C03639=1044.322,83.041,413.959,170.198,36.682,156.905
C03640=1044.329,83.290,413.941,170.200,36.684,156.905
C03641=1044.335,83.539,413.922,170.201,36.685,156.905
C03642=1044.341,83.788,413.904,170.203,36.687,156.906
C03643=1044.347,84.037,413.885,170.205,36.688,156.906
C03644=1044.353,84.287,413.866,170.206,36.689,156.906
C03645=1044.359,84.536,413.848,170.208,36.690,156.906
C03646=1044.366,84.785,413.829,170.211,36.692,156.906
C03647=1044.372,85.034,413.811,170.212,36.693,156.907
C03648=1044.378,85.284,413.791,170.214,36.694,156.907
C03649=1044.384,85.533,413.773,170.216,36.695,156.907
C03650=1044.391,85.782,413.754,170.217,36.697,156.907
C03651=1044.397,86.031,413.735,170.219,36.699,156.908
C03652=1044.403,86.280,413.716,170.222,36.700,156.908
C03653=1044.409,86.529,413.697,170.223,36.701,156.908
C03654=1044.416,86.779,413.679,170.225,36.702,156.909
C03655=1044.422,87.028,413.660,170.227,36.704,156.909
C03656=1044.428,87.277,413.641,170.229,36.705,156.909
C03657=1044.434,87.526,413.622,170.230,36.706,156.909
C03658=1044.440,87.775,413.604,170.233,36.707,156.909
C03659=1044.447,88.024,413.585,170.235,36.709,156.910
C03660=1044.453,88.274,413.566,170.236,36.710,156.910
C03661=1044.459,88.523,413.547,170.238,36.711,156.910
C03662=1044.466,88.773,413.528,170.240,36.712,156.910
C03663=1044.472,89.022,413.509,170.241,36.713,156.911
C03664=1044.479,89.271,413.491,170.243,36.715,156.911
C03665=1044.485,89.521,413.471,170.246,36.717,156.911
C03666=1044.491,89.770,413.453,170.248,36.718,156.912
C03667=1044.497,90.019,413.434,170.249,36.719,156.912
C03668=1044.504,90.268,413.416,170.251,36.720,156.912
C03669=1044.510,90.517,413.396,170.253,36.722,156.912
C03670=1044.516,90.766,413.376,170.254,36.723,156.913
C03671=1044.522,91.015,413.358,170.257,36.724,156.913
C03672=1044.528,91.265,413.338,170.259,36.726,156.913
C03673=1044.534,91.514,413.320,170.260,36.727,156.913
C03674=1044.540,91.763,413.301,170.262,36.728,156.914
C03675=1044.547,92.012,413.281,170.264,36.730,156.914
C03676=1044.552,92.261,413.262,170.265,36.731,156.914
C03677=1044.559,92.510,413.243,170.268,36.733,156.914
C03678=1044.564,92.760,413.224,170.270,36.734,156.915
C03679=1044.572,93.045,413.202,170.272,36.735,156.915
C03680=1044.579,93.332,413.180,170.274,36.737,156.915
C03681=1044.586,93.617,413.158,170.276,36.738,156.916
C03682=1044.593,93.904,413.136,170.278,36.740,156.916
C03683=1044.599,94.153,413.117,170.280,36.741,156.916
C03684=1044.606,94.402,413.098,170.282,36.743,156.916
C03685=1044.612,94.651,413.078,170.284,36.744,156.917
C03686=1044.618,94.900,413.060,170.285,36.745,156.917
C03687=1044.624,95.150,413.040,170.287,36.747,156.917
C03688=1044.630,95.398,413.021,170.290,36.748,156.917
C03689=1044.636,95.648,413.002,170.291,36.749,156.918
C03690=1044.643,95.897,412.983,170.293,36.751,156.918
C03691=1044.649,96.146,412.963,170.295,36.752,156.918
C03692=1044.655,96.396,412.944,170.296,36.753,156.918
C03693=1044.661,96.645,412.925,170.298,36.755,156.919
C03694=1044.667,96.894,412.905,170.301,36.756,156.919
C03695=1044.674,97.143,412.886,170.302,36.758,156.919
C03696=1044.679,97.392,412.867,170.304,36.759,156.920
C03697=1044.686,97.641,412.848,170.306,36.760,156.920
C03698=1044.692,97.891,412.828,170.308,36.761,156.920
C03699=1044.699,98.140,412.809,170.309,36.763,156.920
C03700=1044.705,98.389,412.789,170.312,36.764,156.921
C03701=1044.710,98.638,412.770,170.314,36.766,156.921
C03702=1044.717,98.887,412.751,170.315,36.767,156.921
C03703=1044.723,99.136,412.732,170.317,36.768,156.921
C03704=1044.730,99.386,412.713,170.319,36.769,156.922
C03705=1044.736,99.635,412.693,170.321,36.771,156.922
C03706=1044.742,99.884,412.674,170.322,36.772,156.922
C03707=1044.748,100.133,412.654,170.325,36.774,156.922
C03708=1044.755,100.382,412.635,170.327,36.775,156.923
C03709=1044.761,100.631,412.615,170.328,36.776,156.923
C03710=1044.767,100.881,412.596,170.330,36.777,156.923
C03711=1044.773,101.130,412.576,170.332,36.779,156.923
C03712=1044.779,101.379,412.557,170.334,36.780,156.924
C03713=1044.785,101.628,412.537,170.336,36.782,156.924
C03714=1044.791,101.877,412.518,170.338,36.783,156.924
C03715=1044.798,102.127,412.498,170.340,36.785,156.925
C03716=1044.803,102.376,412.478,170.341,36.786,156.925
C03717=1044.809,102.625,412.458,170.343,36.787,156.925
C03718=1044.816,102.874,412.440,170.346,36.788,156.925
C03719=1044.822,103.123,412.420,170.347,36.790,156.926
C03720=1044.828,103.372,412.400,170.349,36.792,156.926
C03721=1044.834,103.622,412.380,170.351,36.793,156.926
C03722=1044.840,103.870,412.360,170.352,36.794,156.926
C03723=1044.846,104.120,412.341,170.354,36.796,156.927
C03724=1044.853,104.368,412.322,170.357,36.797,156.927
C03725=1044.859,104.618,412.301,170.359,36.798,156.927
C03726=1044.865,104.867,412.282,170.360,36.800,156.928
C03727=1044.871,105.116,412.262,170.362,36.801,156.928
C03728=1044.877,105.365,412.242,170.364,36.803,156.928
C03729=1044.883,105.615,412.223,170.365,36.804,156.928
C03730=1044.890,105.864,412.203,170.368,36.805,156.929
C03731=1044.896,106.112,412.183,170.370,36.807,156.929
C03732=1044.901,106.362,412.164,170.371,36.808,156.929
C03733=1044.908,106.611,412.144,170.373,36.810,156.929
C03734=1044.914,106.860,412.124,170.375,36.811,156.930
C03735=1044.920,107.110,412.105,170.377,36.812,156.930
C03736=1044.927,107.358,412.085,170.379,36.814,156.930
C03737=1044.933,107.608,412.065,170.381,36.815,156.931
C03738=1044.939,107.857,412.046,170.383,36.816,156.931
C03739=1044.945,108.106,412.026,170.385,36.818,156.931
C03740=1044.951,108.355,412.005,170.386,36.819,156.931
C03741=1044.957,108.604,411.985,170.389,36.821,156.932
C03742=1044.963,108.854,411.966,170.391,36.822,156.932
C03743=1044.971,109.139,411.944,170.393,36.824,156.932
C03744=1044.977,109.425,411.921,170.395,36.825,156.933
C03745=1044.986,109.711,411.897,170.397,36.827,156.933
C03746=1044.992,109.997,411.874,170.400,36.828,156.933
C03747=1044.998,110.247,411.855,170.401,36.829,156.933
C03748=1045.005,110.495,411.836,170.403,36.831,156.934
C03749=1045.011,110.745,411.816,170.405,36.832,156.934
C03750=1045.017,110.993,411.796,170.407,36.834,156.934
C03751=1045.023,111.242,411.776,170.408,36.835,156.934
C03752=1045.030,111.492,411.755,170.411,36.837,156.935
C03753=1045.036,111.741,411.736,170.413,36.838,156.935
C03754=1045.042,111.990,411.716,170.414,36.839,156.935
C03755=1045.048,112.240,411.696,170.416,36.840,156.936
C03756=1045.054,112.488,411.676,170.418,36.842,156.936
C03757=1045.060,112.737,411.656,170.420,36.843,156.936
C03758=1045.067,112.987,411.636,170.422,36.845,156.936
C03759=1045.073,113.235,411.616,170.424,36.847,156.937
C03760=1045.078,113.485,411.595,170.426,36.848,156.937
C03761=1045.085,113.734,411.575,170.428,36.849,156.937
C03762=1045.091,113.983,411.555,170.429,36.851,156.938
C03763=1045.097,114.232,411.535,170.432,36.852,156.938
C03764=1045.103,114.481,411.514,170.434,36.853,156.938
C03765=1045.108,114.730,411.494,170.435,36.855,156.939
C03766=1045.114,114.979,411.474,170.437,36.856,156.939
C03767=1045.121,115.229,411.454,170.439,36.858,156.939
C03768=1045.127,115.478,411.434,170.442,36.859,156.939
C03769=1045.132,115.727,411.413,170.443,36.861,156.940
C03770=1045.139,115.976,411.393,170.445,36.863,156.940
C03771=1045.145,116.225,411.373,170.447,36.864,156.940
C03772=1045.150,116.474,411.352,170.448,36.866,156.941
C03773=1045.157,116.724,411.332,170.450,36.867,156.941
C03774=1045.163,116.972,411.312,170.453,36.868,156.941
C03775=1045.169,117.222,411.292,170.455,36.870,156.941
C03776=1045.175,117.471,411.271,170.456,36.871,156.942
C03777=1045.181,117.719,411.250,170.458,36.873,156.942
C03778=1045.187,117.969,411.230,170.460,36.874,156.942
C03779=1045.193,118.218,411.210,170.463,36.875,156.943
C03780=1045.199,118.467,411.190,170.464,36.877,156.943
C03781=1045.205,118.716,411.169,170.466,36.879,156.943
C03782=1045.211,118.965,411.149,170.468,36.880,156.943
C03783=1045.217,119.215,411.128,170.470,36.882,156.944
C03784=1045.223,119.463,411.108,170.472,36.883,156.944
C03785=1045.229,119.712,411.088,170.474,36.885,156.944
C03786=1045.235,119.962,411.067,170.476,36.886,156.945
C03787=1045.241,120.210,411.047,170.477,36.887,156.945
C03788=1045.248,120.460,411.027,170.479,36.889,156.945
C03789=1045.253,120.709,411.006,170.482,36.890,156.945
C03790=1045.260,120.958,410.985,170.484,36.891,156.946
C03791=1045.266,121.207,410.965,170.485,36.893,156.946
C03792=1045.271,121.456,410.944,170.487,36.895,156.946
C03793=1045.278,121.705,410.924,170.489,36.896,156.947
C03794=1045.284,121.954,410.903,170.491,36.898,156.947
C03795=1045.291,122.203,410.883,170.494,36.899,156.947
C03796=1045.296,122.452,410.863,170.495,36.901,156.948
C03797=1045.303,122.702,410.842,170.497,36.902,156.948
C03798=1045.309,122.950,410.822,170.499,36.903,156.948
C03799=1045.315,123.200,410.801,170.501,36.905,156.948
C03800=1045.321,123.449,410.781,170.503,36.906,156.949
C03801=1045.328,123.698,410.760,170.505,36.907,156.949
C03802=1045.333,123.947,410.739,170.507,36.909,156.949
C03803=1045.339,124.196,410.719,170.509,36.910,156.950
C03804=1045.346,124.444,410.698,170.510,36.912,156.950
C03805=1045.352,124.694,410.677,170.513,36.914,156.950
C03806=1045.358,124.943,410.657,170.515,36.915,156.950
C03807=1045.365,125.229,410.633,170.517,36.917,156.951
C03808=1045.372,125.515,410.610,170.519,36.918,156.951
C03809=1045.379,125.801,410.587,170.521,36.920,156.951
C03810=1045.387,126.087,410.563,170.524,36.922,156.952
C03811=1045.392,126.335,410.541,170.526,36.923,156.952
C03812=1045.399,126.585,410.521,170.528,36.925,156.952
C03813=1045.405,126.833,410.501,170.530,36.926,156.953
C03814=1045.411,127.083,410.479,170.531,36.927,156.953
C03815=1045.417,127.332,410.459,170.534,36.929,156.953
C03816=1045.423,127.581,410.438,170.536,36.930,156.953
C03817=1045.430,127.830,410.417,170.538,36.931,156.954
C03818=1045.436,128.078,410.397,170.540,36.933,156.954
C03819=1045.442,128.328,410.376,170.541,36.934,156.954
C03820=1045.448,128.577,410.356,170.543,36.936,156.955
C03821=1045.455,128.826,410.335,170.546,36.937,156.955
C03822=1045.461,129.076,410.314,170.548,36.939,156.955
C03823=1045.467,129.324,410.293,170.550,36.940,156.955
C03824=1045.473,129.573,410.273,170.551,36.942,156.956
C03825=1045.480,129.823,410.251,170.553,36.943,156.956
C03826=1045.486,130.071,410.231,170.556,36.944,156.956
C03827=1045.492,130.321,410.210,170.558,36.946,156.957
C03828=1045.498,130.569,410.190,170.560,36.947,156.957
C03829=1045.505,130.818,410.169,170.561,36.948,156.957
C03830=1045.511,131.068,410.148,170.563,36.950,156.958
C03831=1045.517,131.316,410.127,170.566,36.951,156.958
C03832=1045.523,131.566,410.105,170.568,36.953,156.958
C03833=1045.530,131.815,410.085,170.570,36.955,156.958
C03834=1045.535,132.064,410.064,170.571,36.956,156.959
C03835=1045.541,132.313,410.043,170.573,36.958,156.959
C03836=1045.547,132.562,410.022,170.576,36.959,156.959
C03837=1045.553,132.811,410.001,170.578,36.961,156.960
C03838=1045.559,133.061,409.980,170.580,36.962,156.960
C03839=1045.566,133.309,409.959,170.581,36.964,156.960
C03840=1045.572,133.558,409.937,170.583,36.965,156.960
C03841=1045.578,133.808,409.917,170.586,36.967,156.961
C03842=1045.583,134.056,409.895,170.588,36.968,156.961
C03843=1045.590,134.305,409.874,170.590,36.970,156.961
C03844=1045.596,134.554,409.853,170.591,36.971,156.962
C03845=1045.602,134.804,409.832,170.593,36.973,156.962
C03846=1045.608,135.053,409.811,170.596,36.974,156.962
C03847=1045.614,135.301,409.790,170.598,36.976,156.963
C03848=1045.620,135.550,409.768,170.600,36.977,156.963
C03849=1045.627,135.800,409.748,170.602,36.978,156.963
C03850=1045.632,136.048,409.726,170.603,36.980,156.964
C03851=1045.638,136.297,409.705,170.606,36.981,156.964
C03852=1045.645,136.546,409.684,170.608,36.983,156.964
C03853=1045.651,136.795,409.663,170.610,36.984,156.964
C03854=1045.657,137.045,409.642,170.612,36.986,156.965
C03855=1045.664,137.294,409.621,170.614,36.988,156.965
C03856=1045.670,137.543,409.599,170.616,36.989,156.965
C03857=1045.675,137.791,409.578,170.618,36.991,156.966
C03858=1045.681,138.041,409.557,170.620,36.992,156.966
C03859=1045.687,138.290,409.535,170.622,36.994,156.966
C03860=1045.694,138.539,409.514,170.624,36.995,156.967
C03861=1045.700,138.788,409.493,170.627,36.997,156.967
C03862=1045.706,139.037,409.471,170.628,36.999,156.967
C03863=1045.712,139.285,409.450,170.630,37.000,156.968
C03864=1045.719,139.534,409.429,170.632,37.002,156.968
C03865=1045.725,139.784,409.407,170.634,37.003,156.968
C03866=1045.731,140.033,409.386,170.637,37.005,156.969
C03867=1045.735,140.250,409.368,170.638,37.006,156.969
C03868=1045.741,140.467,409.348,170.640,37.007,156.969
C03869=1045.746,140.685,409.329,170.642,37.009,156.969
C03870=1045.751,140.902,409.311,170.643,37.010,156.970
C03871=1045.757,141.119,409.293,170.646,37.011,156.970
C03872=1045.762,141.336,409.273,170.647,37.013,156.970
C03873=1045.767,141.554,409.255,170.649,37.014,156.971
C03874=1045.772,141.771,409.236,170.651,37.016,156.971
C03875=1045.782,142.171,409.201,170.655,37.018,156.971
C03876=1045.788,142.420,409.180,170.656,37.020,156.972
C03877=1045.794,142.669,409.158,170.658,37.021,156.972
C03878=1045.800,142.918,409.136,170.660,37.023,156.972
C03879=1045.806,143.167,409.115,170.662,37.024,156.973
C03880=1045.813,143.416,409.094,170.665,37.026,156.973
C03881=1045.819,143.665,409.072,170.667,37.027,156.973
C03882=1045.825,143.914,409.051,170.669,37.029,156.973
C03883=1045.831,144.163,409.029,170.670,37.030,156.974
C03884=1045.837,144.412,409.008,170.672,37.032,156.974
C03885=1045.843,144.661,408.986,170.675,37.034,156.974
C03886=1045.849,144.910,408.965,170.677,37.035,156.975
C03887=1045.855,145.160,408.943,170.679,37.037,156.975
C03888=1045.862,145.408,408.921,170.681,37.038,156.975
C03889=1045.867,145.657,408.899,170.684,37.040,156.976
C03890=1045.874,145.906,408.878,170.685,37.041,156.976
C03891=1045.880,146.155,408.856,170.687,37.043,156.976
C03892=1045.886,146.404,408.834,170.689,37.044,156.977
C03893=1045.892,146.654,408.813,170.691,37.046,156.977
C03894=1045.899,146.902,408.790,170.694,37.048,156.977
C03895=1045.904,147.151,408.769,170.696,37.049,156.978
C03896=1045.910,147.400,408.748,170.698,37.051,156.978
C03897=1045.916,147.649,408.726,170.700,37.052,156.978
C03898=1045.923,147.898,408.704,170.703,37.054,156.979
C03899=1045.929,148.147,408.682,170.704,37.056,156.979
C03900=1045.935,148.396,408.660,170.706,37.057,156.979
C03901=1045.940,148.645,408.638,170.708,37.059,156.980
C03902=1045.946,148.894,408.617,170.710,37.061,156.980
C03903=1045.953,149.143,408.594,170.713,37.062,156.980
C03904=1045.959,149.392,408.573,170.715,37.064,156.981
C03905=1045.965,149.641,408.551,170.717,37.065,156.981
C03906=1045.971,149.890,408.529,170.719,37.067,156.981
C03907=1045.978,150.139,408.507,170.722,37.069,156.982
C03908=1045.983,150.388,408.485,170.723,37.070,156.982
C03909=1045.989,150.636,408.463,170.725,37.072,156.982
C03910=1045.995,150.885,408.441,170.727,37.073,156.983
C03911=1046.001,151.135,408.420,170.729,37.075,156.983
C03912=1046.007,151.384,408.397,170.732,37.076,156.983
C03913=1046.013,151.633,408.375,170.734,37.078,156.984
C03914=1046.020,151.881,408.353,170.736,37.080,156.984
C03915=1046.026,152.131,408.331,170.738,37.081,156.984
C03916=1046.032,152.380,408.309,170.741,37.083,156.985
C03917=1046.038,152.629,408.286,170.743,37.085,156.985
C03918=1046.043,152.877,408.265,170.744,37.086,156.985
C03919=1046.050,153.126,408.243,170.746,37.088,156.986
C03920=1046.056,153.375,408.221,170.748,37.090,156.986
C03921=1046.062,153.624,408.198,170.751,37.091,156.986
C03922=1046.068,153.873,408.177,170.753,37.093,156.987
C03923=1046.074,154.122,408.155,170.755,37.095,156.987
C03924=1046.080,154.371,408.133,170.757,37.096,156.987
C03925=1046.087,154.620,408.111,170.760,37.098,156.988
C03926=1046.092,154.869,408.088,170.762,37.099,156.988
C03927=1046.098,155.118,408.066,170.764,37.101,156.988
C03928=1046.104,155.367,408.044,170.766,37.102,156.989
C03929=1046.111,155.616,408.021,170.769,37.104,156.989
C03930=1046.117,155.865,408.000,170.771,37.106,156.989
C03931=1046.123,156.114,407.977,170.772,37.107,156.990
C03932=1046.129,156.363,407.955,170.774,37.109,156.990
C03933=1046.135,156.611,407.933,170.776,37.111,156.990
C03934=1046.141,156.861,407.910,170.779,37.113,156.991
C03935=1046.147,157.110,407.888,170.781,37.114,156.991
C03936=1046.154,157.395,407.863,170.783,37.116,156.991
C03937=1046.161,157.680,407.837,170.787,37.118,156.992
C03938=1046.167,157.965,407.811,170.789,37.120,156.992
C03939=1046.174,158.250,407.785,170.791,37.122,156.993
C03940=1046.181,158.500,407.764,170.793,37.124,156.993
C03941=1046.187,158.748,407.741,170.795,37.125,156.993
C03942=1046.193,158.997,407.718,170.798,37.127,156.994
C03943=1046.199,159.246,407.697,170.800,37.129,156.994
C03944=1046.205,159.495,407.674,170.802,37.130,156.994
C03945=1046.211,159.744,407.652,170.804,37.132,156.995
C03946=1046.218,159.992,407.629,170.807,37.133,156.995
C03947=1046.223,160.242,407.607,170.809,37.135,156.995
C03948=1046.230,160.490,407.585,170.811,37.137,156.996
C03949=1046.235,160.739,407.562,170.813,37.139,156.996
C03950=1046.241,160.988,407.539,170.816,37.141,156.996
C03951=1046.246,161.238,407.516,170.818,37.142,156.997
C03952=1046.253,161.486,407.494,170.820,37.144,156.997
C03953=1046.259,161.735,407.471,170.822,37.145,156.997
C03954=1046.264,161.984,407.448,170.824,37.147,156.998
C03955=1046.270,162.233,407.425,170.826,37.149,156.998
C03956=1046.277,162.482,407.403,170.828,37.151,156.999
C03957=1046.282,162.731,407.380,170.830,37.153,156.999
C03958=1046.288,162.980,407.358,170.833,37.155,156.999
C03959=1046.293,163.229,407.335,170.835,37.156,157.000
C03960=1046.299,163.478,407.312,170.837,37.158,157.000
C03961=1046.306,163.726,407.290,170.839,37.160,157.000
C03962=1046.311,163.975,407.267,170.842,37.162,157.001
C03963=1046.317,164.224,407.244,170.844,37.164,157.001
C03964=1046.323,164.473,407.221,170.846,37.165,157.002
C03965=1046.329,164.722,407.198,170.848,37.167,157.002
C03966=1046.335,164.971,407.175,170.851,37.169,157.002
C03967=1046.341,165.219,407.152,170.853,37.171,157.003
C03968=1046.347,165.469,407.129,170.855,37.173,157.003
C03969=1046.353,165.718,407.106,170.858,37.174,157.003
C03970=1046.359,165.967,407.083,170.860,37.176,157.004
C03971=1046.365,166.215,407.061,170.862,37.178,157.004
C03972=1046.371,166.464,407.038,170.864,37.180,157.005
C03973=1046.376,166.713,407.015,170.867,37.182,157.005
C03974=1046.382,166.962,406.992,170.869,37.184,157.005
C03975=1046.388,167.211,406.969,170.871,37.185,157.006
C03976=1046.394,167.460,406.947,170.873,37.187,157.006
C03977=1046.400,167.709,406.924,170.876,37.189,157.007
C03978=1046.406,167.957,406.901,170.878,37.191,157.007
C03979=1046.413,168.206,406.877,170.880,37.193,157.007
C03980=1046.418,168.455,406.854,170.882,37.194,157.008
C03981=1046.424,168.704,406.831,170.885,37.196,157.008
C03982=1046.430,168.953,406.809,170.887,37.197,157.008
C03983=1046.436,169.202,406.786,170.889,37.199,157.009
C03984=1046.442,169.451,406.763,170.891,37.201,157.009
C03985=1046.448,169.699,406.740,170.894,37.203,157.009
C03986=1046.454,169.949,406.716,170.896,37.205,157.010
C03987=1046.460,170.197,406.693,170.898,37.206,157.010
C03988=1046.466,170.446,406.670,170.900,37.208,157.011
C03989=1046.472,170.695,406.647,170.903,37.210,157.011
C03990=1046.478,170.944,406.625,170.905,37.212,157.011
C03991=1046.484,171.193,406.601,170.907,37.214,157.012
C03992=1046.490,171.442,406.578,170.909,37.215,157.012
C03993=1046.496,171.691,406.555,170.912,37.217,157.012
C03994=1046.503,171.939,406.532,170.914,37.219,157.013
C03995=1046.508,172.188,406.509,170.916,37.221,157.013
C03996=1046.515,172.437,406.485,170.919,37.223,157.014
C03997=1046.521,172.686,406.462,170.921,37.224,157.014
C03998=1046.526,172.935,406.439,170.923,37.226,157.014
C03999=1046.532,173.184,406.416,170.925,37.228,157.015
C04000=1046.540,173.468,406.390,170.929,37.231,157.015
C04001=1046.547,173.754,406.363,170.931,37.232,157.016
C04002=1046.554,174.038,406.337,170.934,37.234,157.016
C04003=1046.561,174.323,406.310,170.937,37.237,157.016
C04004=1046.566,174.572,406.287,170.939,37.238,157.017
C04005=1046.572,174.820,406.263,170.941,37.240,157.017
C04006=1046.579,175.070,406.240,170.943,37.242,157.018
C04007=1046.584,175.319,406.217,170.946,37.244,157.018
C04008=1046.591,175.567,406.194,170.948,37.246,157.018
C04009=1046.597,175.816,406.171,170.950,37.247,157.019
C04010=1046.604,176.064,406.147,170.953,37.249,157.019
C04011=1046.609,176.313,406.124,170.956,37.251,157.020
C04012=1046.616,176.563,406.101,170.958,37.253,157.020
C04013=1046.622,176.811,406.077,170.960,37.255,157.020
C04014=1046.627,177.060,406.054,170.963,37.256,157.021
C04015=1046.634,177.309,406.030,170.965,37.258,157.021
C04016=1046.640,177.558,406.007,170.967,37.260,157.021
C04017=1046.646,177.806,405.984,170.969,37.262,157.022
C04018=1046.653,178.056,405.961,170.972,37.264,157.022
C04019=1046.659,178.304,405.937,170.974,37.265,157.023
C04020=1046.665,178.553,405.914,170.977,37.267,157.023
C04021=1046.671,178.802,405.890,170.979,37.269,157.023
C04022=1046.677,179.051,405.867,170.982,37.271,157.024
C04023=1046.684,179.300,405.843,170.984,37.273,157.024
C04024=1046.689,179.549,405.820,170.986,37.274,157.024
C04025=1046.695,179.797,405.797,170.988,37.276,157.025
C04026=1046.702,180.046,405.773,170.991,37.278,157.025
C04027=1046.708,180.295,405.750,170.994,37.280,157.026
C04028=1046.714,180.544,405.726,170.996,37.281,157.026
C04029=1046.720,180.793,405.703,170.999,37.283,157.026
C04030=1046.727,181.041,405.679,171.001,37.285,157.027
C04031=1046.733,181.290,405.656,171.003,37.287,157.027
C04032=1046.739,181.538,405.633,171.005,37.289,157.027
C04033=1046.746,181.788,405.609,171.008,37.290,157.028
C04034=1046.752,182.036,405.586,171.011,37.292,157.028
C04035=1046.758,182.285,405.562,171.013,37.295,157.029
C04036=1046.764,182.534,405.539,171.016,37.296,157.029
C04037=1046.771,182.783,405.515,171.018,37.298,157.030
C04038=1046.777,183.031,405.491,171.020,37.300,157.030
C04039=1046.783,183.281,405.468,171.022,37.302,157.030
C04040=1046.789,183.529,405.444,171.026,37.304,157.031
C04041=1046.796,183.778,405.420,171.028,37.305,157.031
C04042=1046.801,184.027,405.397,171.030,37.307,157.031
C04043=1046.807,184.276,405.372,171.032,37.309,157.032
C04044=1046.813,184.525,405.349,171.035,37.311,157.032
C04045=1046.819,184.773,405.325,171.037,37.313,157.033
C04046=1046.825,185.022,405.301,171.039,37.315,157.033
C04047=1046.831,185.271,405.277,171.043,37.317,157.034
C04048=1046.837,185.520,405.252,171.045,37.319,157.034
C04049=1046.843,185.769,405.229,171.047,37.322,157.034
C04050=1046.848,186.017,405.205,171.050,37.323,157.035
C04051=1046.855,186.266,405.181,171.052,37.325,157.035
C04052=1046.860,186.515,405.157,171.054,37.328,157.036
C04053=1046.867,186.764,405.133,171.057,37.329,157.036
C04054=1046.872,187.012,405.108,171.060,37.331,157.037
C04055=1046.879,187.261,405.084,171.062,37.334,157.037
C04056=1046.884,187.510,405.060,171.064,37.335,157.037
C04057=1046.890,187.758,405.037,171.067,37.338,157.038
C04058=1046.896,188.008,405.012,171.069,37.340,157.038
C04059=1046.902,188.256,404.988,171.071,37.341,157.039
C04060=1046.908,188.505,404.964,171.075,37.344,157.039
C04061=1046.914,188.753,404.940,171.077,37.346,157.040
C04062=1046.920,189.003,404.915,171.079,37.347,157.040
C04063=1046.926,189.251,404.892,171.082,37.350,157.040
C04064=1046.933,189.535,404.864,171.085,37.352,157.041
C04065=1046.940,189.820,404.836,171.087,37.354,157.041
C04066=1046.946,190.105,404.809,171.091,37.356,157.042
C04067=1046.953,190.389,404.781,171.093,37.359,157.042
C04068=1046.960,190.638,404.757,171.095,37.361,157.043
C04069=1046.965,190.886,404.732,171.098,37.363,157.043
C04070=1046.971,191.136,404.708,171.101,37.365,157.044
C04071=1046.977,191.384,404.684,171.103,37.367,157.044
C04072=1046.983,191.633,404.659,171.106,37.369,157.045
C04073=1046.990,191.881,404.635,171.108,37.371,157.045
C04074=1046.995,192.130,404.610,171.111,37.373,157.045
C04075=1047.002,192.379,404.586,171.114,37.375,157.046
C04076=1047.007,192.628,404.562,171.116,37.377,157.046
C04077=1047.014,192.877,404.538,171.118,37.380,157.047
C04078=1047.019,193.125,404.514,171.120,37.381,157.047
C04079=1047.026,193.374,404.489,171.124,37.383,157.048
C04080=1047.032,193.623,404.464,171.126,37.386,157.048
C04081=1047.038,193.871,404.441,171.128,37.387,157.049
C04082=1047.044,194.120,404.416,171.131,37.390,157.049
C04083=1047.050,194.368,404.392,171.134,37.391,157.049
C04084=1047.056,194.617,404.367,171.136,37.394,157.050
C04085=1047.062,194.867,404.343,171.139,37.396,157.050
C04086=1047.068,195.115,404.319,171.141,37.397,157.051
C04087=1047.074,195.364,404.294,171.144,37.400,157.051
C04088=1047.081,195.613,404.270,171.147,37.402,157.052
C04089=1047.086,195.861,404.245,171.149,37.404,157.052
C04090=1047.093,196.110,404.221,171.151,37.406,157.052
C04091=1047.099,196.359,404.196,171.155,37.408,157.053
C04092=1047.105,196.607,404.172,171.157,37.410,157.053
C04093=1047.111,196.856,404.147,171.159,37.412,157.054
C04094=1047.117,197.105,404.122,171.162,37.414,157.054
C04095=1047.124,197.353,404.098,171.165,37.416,157.055
C04096=1047.130,197.602,404.073,171.167,37.418,157.055
C04097=1047.136,197.851,404.049,171.170,37.421,157.056
C04098=1047.142,198.100,404.024,171.173,37.422,157.056
C04099=1047.148,198.348,404.000,171.175,37.425,157.057
C04100=1047.155,198.597,403.975,171.178,37.427,157.057
C04101=1047.161,198.846,403.950,171.181,37.429,157.057
C04102=1047.168,199.094,403.926,171.183,37.431,157.058
C04103=1047.173,199.343,403.901,171.186,37.433,157.058
C04104=1047.179,199.592,403.877,171.188,37.435,157.059
C04105=1047.186,199.841,403.852,171.191,37.437,157.059
C04106=1047.192,200.090,403.827,171.193,37.439,157.060
C04107=1047.199,200.338,403.803,171.196,37.441,157.060
C04108=1047.204,200.587,403.778,171.199,37.443,157.061
C04109=1047.211,200.835,403.754,171.202,37.446,157.061
C04110=1047.217,201.084,403.728,171.204,37.447,157.061
C04111=1047.223,201.333,403.704,171.207,37.450,157.062
C04112=1047.229,201.582,403.678,171.210,37.452,157.063
C04113=1047.235,201.830,403.655,171.212,37.454,157.063
C04114=1047.241,202.079,403.629,171.215,37.456,157.063
C04115=1047.248,202.327,403.604,171.218,37.459,157.064
C04116=1047.253,202.577,403.579,171.220,37.460,157.064
C04117=1047.259,202.825,403.554,171.223,37.463,157.065
C04118=1047.265,203.073,403.529,171.226,37.465,157.065
C04119=1047.271,203.323,403.504,171.228,37.468,157.066
C04120=1047.277,203.571,403.479,171.230,37.469,157.066
C04121=1047.284,203.820,403.454,171.234,37.472,157.067
C04122=1047.289,204.068,403.429,171.236,37.474,157.067
C04123=1047.295,204.317,403.404,171.238,37.476,157.068
C04124=1047.301,204.566,403.379,171.242,37.478,157.068
C04125=1047.307,204.814,403.353,171.244,37.481,157.069
C04126=1047.314,205.063,403.329,171.247,37.483,157.069
C04127=1047.321,205.312,403.303,171.250,37.485,157.070
C04128=1047.346,206.364,403.197,171.496,37.584,157.093
C04129=1047.353,206.631,403.169,171.497,37.587,157.094
C04130=1047.360,206.899,403.141,171.500,37.590,157.094
C04131=1047.367,207.167,403.113,171.502,37.594,157.095
C04132=1047.375,207.435,403.084,171.504,37.597,157.096
C04133=1047.381,207.684,403.059,171.506,37.600,157.096
C04134=1047.387,207.932,403.032,171.509,37.603,157.097
C04135=1047.394,208.181,403.006,171.510,37.606,157.098
C04136=1047.400,208.429,402.980,171.513,37.609,157.098
C04137=1047.407,208.678,402.953,171.514,37.612,157.099
C04138=1047.413,208.926,402.927,171.517,37.615,157.099
C04139=1047.420,209.175,402.900,171.518,37.618,157.100
C04140=1047.426,209.423,402.875,171.521,37.621,157.101
C04141=1047.433,209.672,402.848,171.522,37.624,157.101
C04142=1047.439,209.920,402.822,171.525,37.627,157.102
C04143=1047.445,210.169,402.795,171.527,37.630,157.103
C04144=1047.452,210.417,402.769,171.529,37.633,157.103
C04145=1047.459,210.666,402.743,171.531,37.636,157.104
C04146=1047.465,210.915,402.716,171.533,37.639,157.105
C04147=1047.472,211.163,402.690,171.535,37.642,157.105
C04148=1047.479,211.411,402.663,171.538,37.645,157.106
C04149=1047.484,211.660,402.637,171.539,37.648,157.107
C04150=1047.492,211.909,402.610,171.542,37.651,157.107
C04151=1047.497,212.157,402.583,171.543,37.654,157.108
C04152=1047.504,212.406,402.557,171.546,37.657,157.109
C04153=1047.510,212.654,402.530,171.547,37.660,157.109
C04154=1047.517,212.903,402.504,171.550,37.663,157.110
C04155=1047.523,213.151,402.477,171.552,37.666,157.111
C04156=1047.530,213.400,402.451,171.554,37.669,157.111
C04157=1047.536,213.648,402.424,171.556,37.672,157.112
C04158=1047.543,213.897,402.397,171.558,37.675,157.113
C04159=1047.549,214.145,402.370,171.560,37.678,157.113
C04160=1047.556,214.394,402.343,171.563,37.681,157.114
C04161=1047.562,214.642,402.317,171.564,37.684,157.114
C04162=1047.568,214.891,402.290,171.567,37.687,157.115
C04163=1047.575,215.139,402.264,171.569,37.690,157.116
C04164=1047.581,215.388,402.237,171.571,37.693,157.116
C04165=1047.587,215.636,402.210,171.573,37.696,157.117
C04166=1047.594,215.884,402.184,171.575,37.699,157.118
C04167=1047.600,216.133,402.157,171.577,37.702,157.118
C04168=1047.607,216.382,402.130,171.580,37.705,157.119
C04169=1047.614,216.631,402.103,171.581,37.708,157.120
C04170=1047.621,216.878,402.077,171.584,37.711,157.120
C04171=1047.627,217.127,402.050,171.586,37.714,157.121
C04172=1047.633,217.375,402.023,171.588,37.717,157.122
C04173=1047.640,217.624,401.997,171.590,37.720,157.122
C04174=1047.646,217.872,401.969,171.593,37.723,157.123
C04175=1047.653,218.121,401.943,171.594,37.726,157.124
C04176=1047.659,218.370,401.916,171.597,37.728,157.124
C04177=1047.665,218.618,401.888,171.599,37.731,157.125
C04178=1047.673,218.866,401.862,171.601,37.734,157.125
C04179=1047.679,219.115,401.835,171.603,37.737,157.126
C04180=1047.685,219.363,401.809,171.606,37.740,157.127
C04181=1047.692,219.612,401.781,171.607,37.743,157.127
C04182=1047.698,219.860,401.755,171.610,37.746,157.128
C04183=1047.705,220.108,401.727,171.612,37.749,157.129
C04184=1047.712,220.357,401.700,171.614,37.752,157.129
C04185=1047.720,220.631,401.671,171.616,37.756,157.130
C04186=1047.726,220.904,401.641,171.619,37.759,157.131
C04187=1047.733,221.177,401.611,171.621,37.762,157.132
C04188=1047.740,221.451,401.581,171.624,37.765,157.132
C04189=1047.746,221.699,401.555,171.626,37.768,157.133
C04190=1047.753,221.948,401.527,171.628,37.771,157.133
C04191=1047.759,222.197,401.500,171.630,37.774,157.134
C04192=1047.766,222.444,401.473,171.633,37.777,157.135
C04193=1047.772,222.693,401.446,171.634,37.780,157.135
C04194=1047.778,222.941,401.419,171.637,37.783,157.136
C04195=1047.785,223.190,401.392,171.639,37.786,157.137
C04196=1047.791,223.438,401.364,171.642,37.789,157.137
C04197=1047.797,223.687,401.337,171.643,37.792,157.138
C04198=1047.804,223.935,401.310,171.646,37.795,157.139
C04199=1047.811,224.183,401.282,171.648,37.798,157.139
C04200=1047.818,224.432,401.255,171.650,37.801,157.140
C04201=1047.824,224.680,401.228,171.652,37.804,157.141
C04202=1047.830,224.929,401.201,171.655,37.807,157.141
C04203=1047.837,225.178,401.173,171.657,37.810,157.142
C04204=1047.843,225.425,401.146,171.659,37.813,157.143
C04205=1047.849,225.674,401.119,171.661,37.815,157.143
C04206=1047.856,225.923,401.091,171.664,37.818,157.144
C04207=1047.863,226.171,401.064,171.666,37.821,157.145
C04208=1047.869,226.419,401.037,171.668,37.824,157.145
C04209=1047.876,226.668,401.010,171.670,37.827,157.146
C04210=1047.883,226.916,400.982,171.673,37.830,157.147
C04211=1047.889,227.165,400.955,171.675,37.833,157.147
C04212=1047.895,227.413,400.928,171.677,37.836,157.148
C04213=1047.902,227.661,400.900,171.679,37.839,157.148
C04214=1047.908,227.910,400.873,171.682,37.842,157.149
C04215=1047.915,228.159,400.845,171.685,37.845,157.150
C04216=1047.922,228.407,400.818,171.687,37.847,157.150
C04217=1047.928,228.655,400.791,171.688,37.850,157.151
C04218=1047.935,228.904,400.764,171.691,37.853,157.152
C04219=1047.941,229.152,400.736,171.693,37.856,157.152
C04220=1047.947,229.401,400.708,171.696,37.859,157.153
C04221=1047.954,229.649,400.680,171.698,37.862,157.154
C04222=1047.960,229.897,400.652,171.700,37.865,157.154
C04223=1047.967,230.146,400.625,171.703,37.868,157.155
C04224=1047.973,230.394,400.597,171.705,37.871,157.156
C04225=1047.980,230.643,400.570,171.708,37.874,157.156
C04226=1047.986,230.891,400.543,171.710,37.877,157.157
C04227=1047.992,231.139,400.515,171.712,37.880,157.158
C04228=1047.999,231.388,400.487,171.714,37.883,157.158
C04229=1048.005,231.637,400.459,171.717,37.886,157.159
C04230=1048.012,231.885,400.431,171.719,37.889,157.159
C04231=1048.018,232.133,400.403,171.722,37.891,157.160
C04232=1048.025,232.381,400.376,171.723,37.894,157.161
C04233=1048.031,232.630,400.348,171.726,37.897,157.161
C04234=1048.038,232.878,400.321,171.728,37.900,157.162
C04235=1048.044,233.127,400.292,171.731,37.903,157.163
C04236=1048.051,233.375,400.265,171.733,37.906,157.163
C04237=1048.057,233.624,400.237,171.736,37.909,157.164
C04238=1048.063,233.871,400.209,171.737,37.912,157.165
C04239=1048.069,234.120,400.181,171.740,37.915,157.165
C04240=1048.076,234.369,400.153,171.742,37.918,157.166
C04241=1048.082,234.634,400.123,171.745,37.921,157.167
C04242=1048.090,234.900,400.093,171.747,37.924,157.167
C04243=1048.097,235.166,400.064,171.750,37.927,157.168
C04244=1048.104,235.432,400.034,171.753,37.931,157.169
C04245=1048.110,235.680,400.006,171.755,37.934,157.170
C04246=1048.116,235.929,399.978,171.758,37.937,157.170
C04247=1048.123,236.177,399.950,171.760,37.940,157.171
C04248=1048.129,236.425,399.921,171.762,37.943,157.172
C04249=1048.136,236.674,399.893,171.764,37.945,157.172
C04250=1048.143,236.922,399.866,171.767,37.948,157.173
C04251=1048.149,237.171,399.838,171.769,37.951,157.173
C04252=1048.155,237.419,399.810,171.772,37.954,157.174
C04253=1048.162,237.667,399.781,171.774,37.957,157.175
C04254=1048.169,237.916,399.753,171.777,37.960,157.175
C04255=1048.174,238.164,399.726,171.779,37.963,157.176
C04256=1048.181,238.412,399.698,171.782,37.965,157.177
C04257=1048.188,238.660,399.669,171.783,37.968,157.177
C04258=1048.194,238.909,399.641,171.786,37.971,157.178
C04259=1048.201,239.157,399.613,171.788,37.974,157.179
C04260=1048.208,239.405,399.585,171.791,37.977,157.179
C04261=1048.214,239.654,399.557,171.793,37.980,157.180
C04262=1048.220,239.902,399.529,171.796,37.983,157.181
C04263=1048.227,240.150,399.500,171.799,37.986,157.181
C04264=1048.233,240.399,399.472,171.801,37.989,157.182
C04265=1048.240,240.647,399.444,171.804,37.992,157.183
C04266=1048.246,240.895,399.415,171.806,37.995,157.183
C04267=1048.253,241.144,399.388,171.809,37.998,157.184
C04268=1048.259,241.392,399.360,171.811,38.001,157.185
C04269=1048.266,241.640,399.331,171.814,38.004,157.185
C04270=1048.272,241.889,399.303,171.815,38.006,157.186
C04271=1048.279,242.137,399.274,171.818,38.009,157.187
C04272=1048.285,242.386,399.246,171.820,38.012,157.187
C04273=1048.292,242.633,399.217,171.823,38.015,157.188
C04274=1048.298,242.882,399.189,171.825,38.018,157.189
C04275=1048.305,243.130,399.160,171.828,38.021,157.189
C04276=1048.310,243.379,399.132,171.830,38.024,157.190
C04277=1048.317,243.627,399.103,171.833,38.027,157.191
C04278=1048.323,243.875,399.075,171.835,38.030,157.191
C04279=1048.330,244.123,399.046,171.838,38.033,157.192
C04280=1048.337,244.371,399.018,171.841,38.036,157.193
C04281=1048.343,244.621,398.989,171.843,38.039,157.193
C04282=1048.349,244.869,398.960,171.846,38.042,157.194
C04283=1048.356,245.117,398.932,171.848,38.044,157.195
C04284=1048.362,245.365,398.903,171.851,38.047,157.195
C04285=1048.369,245.613,398.875,171.853,38.050,157.196
C04286=1048.375,245.862,398.847,171.856,38.053,157.197
C04287=1048.382,246.110,398.818,171.858,38.056,157.197
C04288=1048.388,246.358,398.789,171.861,38.059,157.198
C04289=1048.394,246.606,398.759,171.863,38.062,157.199
C04290=1048.400,246.855,398.731,171.866,38.065,157.199
C04291=1048.407,247.103,398.703,171.869,38.068,157.200
C04292=1048.413,247.351,398.674,171.870,38.071,157.201
C04293=1048.419,247.599,398.645,171.873,38.074,157.201
C04294=1048.425,247.848,398.616,171.875,38.077,157.202
C04295=1048.432,248.096,398.587,171.878,38.080,157.203
C04296=1048.438,248.344,398.558,171.880,38.083,157.203
C04297=1048.445,248.605,398.527,171.884,38.086,157.204
C04298=1048.452,248.865,398.498,171.886,38.089,157.205
C04299=1048.459,249.124,398.467,171.889,38.092,157.205
C04300=1048.465,249.385,398.438,171.892,38.095,157.206
C04301=1048.471,249.633,398.409,171.894,38.098,157.207
C04302=1048.478,249.881,398.379,171.897,38.102,157.208
C04303=1048.484,250.129,398.350,171.899,38.104,157.208
C04304=1048.490,250.377,398.321,171.902,38.107,157.209
C04305=1048.497,250.626,398.292,171.904,38.110,157.210
C04306=1048.503,250.874,398.263,171.907,38.113,157.210
C04307=1048.510,251.122,398.234,171.909,38.116,157.211
C04308=1048.517,251.370,398.205,171.912,38.119,157.212
C04309=1048.523,251.618,398.176,171.915,38.122,157.212
C04310=1048.529,251.867,398.148,171.917,38.125,157.213
C04311=1048.536,252.116,398.119,171.920,38.128,157.214
C04312=1048.542,252.364,398.090,171.922,38.131,157.214
C04313=1048.548,252.611,398.060,171.925,38.134,157.215
C04314=1048.555,252.859,398.031,171.927,38.136,157.216
C04315=1048.561,253.108,398.002,171.930,38.139,157.216
C04316=1048.568,253.356,397.972,171.933,38.142,157.217
C04317=1048.574,253.605,397.943,171.936,38.145,157.218
C04318=1048.581,253.852,397.915,171.938,38.148,157.218
C04319=1048.587,254.100,397.886,171.941,38.152,157.219
C04320=1048.594,254.349,397.856,171.944,38.154,157.220
C04321=1048.600,254.597,397.827,171.946,38.157,157.220
C04322=1048.607,254.846,397.798,171.949,38.160,157.221
C04323=1048.613,255.094,397.769,171.951,38.163,157.222
C04324=1048.620,255.343,397.740,171.954,38.166,157.222
C04325=1048.626,255.590,397.710,171.956,38.169,157.223
C04326=1048.633,255.838,397.681,171.959,38.172,157.224
C04327=1048.639,256.087,397.652,171.963,38.175,157.224
C04328=1048.646,256.335,397.623,171.965,38.178,157.225
C04329=1048.652,256.583,397.594,171.968,38.181,157.226
C04330=1048.658,256.831,397.564,171.970,38.183,157.226
C04331=1048.665,257.080,397.535,171.973,38.186,157.227
C04332=1048.672,257.328,397.505,171.975,38.189,157.228
C04333=1048.679,257.576,397.477,171.978,38.192,157.228
C04334=1048.686,257.824,397.447,171.980,38.195,157.229
C04335=1048.692,258.072,397.418,171.984,38.198,157.230
C04336=1048.699,258.321,397.388,171.987,38.201,157.230
C04337=1048.705,258.569,397.359,171.989,38.204,157.231
C04338=1048.712,258.816,397.330,171.992,38.207,157.232
C04339=1048.718,259.065,397.300,171.994,38.209,157.232
C04340=1048.725,259.313,397.271,171.997,38.212,157.233
C04341=1048.731,259.561,397.241,172.000,38.215,157.234
C04342=1048.738,259.810,397.212,172.003,38.218,157.234
C04343=1048.744,260.058,397.183,172.005,38.221,157.235
C04344=1048.751,260.306,397.153,172.008,38.224,157.236
C04345=1048.758,260.554,397.124,172.011,38.227,157.236
C04346=1048.765,260.802,397.094,172.013,38.230,157.237
C04347=1048.771,261.051,397.065,172.017,38.232,157.238
C04348=1048.777,261.299,397.036,172.019,38.235,157.238
C04349=1048.785,261.547,397.006,172.022,38.238,157.239
C04350=1048.791,261.795,396.976,172.024,38.241,157.240
C04351=1048.798,262.043,396.946,172.028,38.244,157.241
C04352=1048.804,262.291,396.917,172.030,38.247,157.241
C04353=1048.811,262.550,396.886,172.033,38.250,157.242
C04354=1048.818,262.809,396.855,172.036,38.253,157.243
C04355=1048.824,263.067,396.825,172.039,38.256,157.243
C04356=1048.832,263.325,396.793,172.042,38.259,157.244
C04357=1048.838,263.573,396.764,172.044,38.262,157.245
C04358=1048.844,263.821,396.733,172.047,38.265,157.245
C04359=1048.851,264.070,396.704,172.050,38.268,157.246
C04360=1048.857,264.317,396.674,172.053,38.271,157.247
C04361=1048.864,264.566,396.643,172.056,38.274,157.248
C04362=1048.870,264.814,396.614,172.058,38.277,157.248
C04363=1048.877,265.062,396.584,172.061,38.280,157.249
C04364=1048.883,265.310,396.554,172.065,38.283,157.250
C04365=1048.890,265.558,396.524,172.067,38.286,157.250
C04366=1048.896,265.806,396.495,172.070,38.289,157.251
C04367=1048.903,266.055,396.464,172.072,38.292,157.252
C04368=1048.909,266.302,396.434,172.075,38.295,157.252
C04369=1048.917,266.551,396.404,172.078,38.298,157.253
C04370=1048.922,266.799,396.375,172.081,38.301,157.254
C04371=1048.929,267.047,396.344,172.084,38.304,157.255
C04372=1048.936,267.295,396.315,172.086,38.307,157.255
C04373=1048.942,267.543,396.284,172.090,38.310,157.256
C04374=1048.949,267.791,396.254,172.092,38.313,157.257
C04375=1048.955,268.039,396.224,172.095,38.315,157.257
C04376=1048.961,268.287,396.194,172.098,38.319,157.258
C04377=1048.969,268.536,396.164,172.101,38.322,157.259
C04378=1048.974,268.784,396.134,172.104,38.325,157.259
C04379=1048.982,269.032,396.104,172.106,38.327,157.260
C04380=1048.987,269.280,396.074,172.110,38.330,157.261
C04381=1048.995,269.528,396.043,172.113,38.334,157.262
C04382=1049.000,269.776,396.013,172.115,38.337,157.262
C04383=1049.007,270.024,395.983,172.118,38.340,157.263
C04384=1049.013,270.272,395.953,172.121,38.342,157.264
C04385=1049.020,270.520,395.922,172.124,38.345,157.264
C04386=1049.027,270.768,395.892,172.127,38.349,157.265
C04387=1049.033,271.016,395.861,172.130,38.352,157.266
C04388=1049.040,271.264,395.831,172.133,38.354,157.266
C04389=1049.046,271.512,395.801,172.135,38.357,157.267
C04390=1049.053,271.760,395.771,172.138,38.361,157.268
C04391=1049.059,272.009,395.740,172.142,38.364,157.269
C04392=1049.066,272.256,395.710,172.144,38.366,157.269
C04393=1049.072,272.505,395.680,172.147,38.369,157.270
C04394=1049.078,272.752,395.649,172.150,38.373,157.271
C04395=1049.086,273.000,395.618,172.153,38.376,157.271
C04396=1049.092,273.249,395.588,172.156,38.379,157.272
C04397=1049.098,273.497,395.557,172.159,38.381,157.273
C04398=1049.105,273.745,395.527,172.162,38.385,157.274
C04399=1049.112,273.993,395.496,172.164,38.388,157.274
C04400=1049.117,274.241,395.465,172.168,38.390,157.275
C04401=1049.125,274.489,395.435,172.171,38.394,157.276
C04402=1049.130,274.737,395.405,172.173,38.397,157.277
C04403=1049.137,274.985,395.374,172.177,38.400,157.277
C04404=1049.144,275.233,395.343,172.179,38.403,157.278
C04405=1049.150,275.481,395.313,172.182,38.406,157.279
C04406=1049.157,275.729,395.282,172.186,38.409,157.279
C04407=1049.163,275.977,395.251,172.188,38.412,157.280
C04408=1049.170,276.225,395.221,172.191,38.415,157.281
C04409=1049.177,276.488,395.187,172.195,38.418,157.282
C04410=1049.184,276.751,395.155,172.197,38.421,157.282
C04411=1049.191,277.013,395.123,172.201,38.425,157.283
C04412=1049.198,277.276,395.091,172.203,38.428,157.284
C04413=1049.204,277.524,395.059,172.207,38.431,157.285
C04414=1049.210,277.772,395.029,172.210,38.434,157.285
C04415=1049.217,278.020,394.998,172.213,38.437,157.286
C04416=1049.224,278.268,394.967,172.216,38.440,157.287
C04417=1049.231,278.516,394.936,172.219,38.443,157.288
C04418=1049.237,278.764,394.906,172.222,38.446,157.288
C04419=1049.243,279.012,394.874,172.225,38.449,157.289
C04420=1049.250,279.260,394.843,172.229,38.452,157.290
C04421=1049.257,279.508,394.812,172.231,38.455,157.290
C04422=1049.262,279.756,394.782,172.234,38.458,157.291
C04423=1049.269,280.004,394.750,172.237,38.461,157.292
C04424=1049.275,280.252,394.720,172.240,38.465,157.293
C04425=1049.282,280.500,394.688,172.244,38.468,157.293
C04426=1049.288,280.747,394.657,172.246,38.470,157.294
C04427=1049.295,280.996,394.626,172.249,38.474,157.295
C04428=1049.301,281.244,394.595,172.253,38.477,157.296
C04429=1049.308,281.492,394.563,172.255,38.480,157.296
C04430=1049.314,281.740,394.533,172.259,38.483,157.297
C04431=1049.321,281.987,394.502,172.262,38.486,157.298
C04432=1049.327,282.235,394.470,172.265,38.489,157.299
C04433=1049.334,282.484,394.440,172.268,38.493,157.299
C04434=1049.341,282.732,394.408,172.270,38.495,157.300
C04435=1049.347,282.980,394.377,172.274,38.498,157.301
C04436=1049.353,283.227,394.346,172.277,38.502,157.302
C04437=1049.360,283.475,394.314,172.280,38.505,157.302
C04438=1049.367,283.723,394.283,172.283,38.508,157.303
C04439=1049.373,283.971,394.252,172.287,38.511,157.304
C04440=1049.380,284.219,394.221,172.289,38.514,157.305
C04441=1049.387,284.467,394.189,172.293,38.517,157.305
C04442=1049.394,284.715,394.158,172.296,38.520,157.306
C04443=1049.400,284.962,394.127,172.299,38.523,157.307
C04444=1049.406,285.211,394.096,172.302,38.527,157.308
C04445=1049.413,285.459,394.065,172.306,38.530,157.308
C04446=1049.419,285.706,394.033,172.308,38.533,157.309
C04447=1049.426,285.954,394.002,172.312,38.536,157.310
C04448=1049.433,286.202,393.970,172.314,38.539,157.311
C04449=1049.440,286.450,393.939,172.318,38.542,157.311
C04450=1049.446,286.698,393.907,172.321,38.545,157.312
C04451=1049.453,286.946,393.876,172.324,38.548,157.313
C04452=1049.459,287.194,393.844,172.327,38.551,157.314
C04453=1049.466,287.442,393.812,172.331,38.554,157.314
C04454=1049.473,287.690,393.781,172.333,38.557,157.315
C04455=1049.479,287.938,393.750,172.337,38.561,157.316
C04456=1049.486,288.186,393.718,172.340,38.564,157.317
C04457=1049.493,288.434,393.687,172.343,38.567,157.317
C04458=1049.499,288.682,393.655,172.346,38.570,157.318
C04459=1049.506,288.929,393.623,172.350,38.573,157.319
C04460=1049.512,289.176,393.591,172.352,38.577,157.320
C04461=1049.519,289.424,393.560,172.356,38.579,157.320
C04462=1049.525,289.673,393.528,172.359,38.583,157.321
C04463=1049.531,289.920,393.497,172.363,38.586,157.322
C04464=1049.538,290.168,393.465,172.366,38.589,157.323
C04465=1049.546,290.443,393.429,172.369,38.592,157.324
C04466=1049.553,290.717,393.395,172.373,38.596,157.325
C04467=1049.560,290.992,393.359,172.376,38.600,157.325
C04468=1049.567,291.265,393.324,172.380,38.603,157.326
C04469=1049.574,291.513,393.292,172.383,38.607,157.327
C04470=1049.580,291.761,393.260,172.386,38.609,157.328
C04471=1049.587,292.009,393.228,172.390,38.613,157.329
C04472=1049.594,292.256,393.197,172.393,38.616,157.329
C04473=1049.600,292.505,393.165,172.397,38.619,157.330
C04474=1049.607,292.752,393.132,172.399,38.622,157.331
C04475=1049.613,293.000,393.101,172.403,38.626,157.332
C04476=1049.620,293.248,393.068,172.407,38.629,157.332
C04477=1049.627,293.496,393.036,172.409,38.632,157.333
C04478=1049.634,293.744,393.005,172.413,38.635,157.334
C04479=1049.640,293.992,392.972,172.416,38.638,157.335
C04480=1049.647,294.239,392.941,172.419,38.642,157.336
C04481=1049.653,294.487,392.908,172.423,38.645,157.336
C04482=1049.660,294.735,392.877,172.426,38.648,157.337
C04483=1049.666,294.983,392.844,172.429,38.651,157.338
C04484=1049.673,295.230,392.812,172.432,38.655,157.339
C04485=1049.680,295.479,392.779,172.436,38.658,157.340
C04486=1049.686,295.727,392.748,172.440,38.661,157.340
C04487=1049.693,295.974,392.715,172.442,38.664,157.341
C04488=1049.700,296.222,392.683,172.446,38.667,157.342
C04489=1049.706,296.470,392.651,172.450,38.671,157.343
C04490=1049.712,296.717,392.618,172.452,38.674,157.344
C04491=1049.718,296.965,392.586,172.456,38.677,157.344
C04492=1049.725,297.213,392.554,172.459,38.680,157.345
C04493=1049.731,297.460,392.521,172.463,38.684,157.346
C04494=1049.738,297.709,392.488,172.466,38.687,157.347
C04495=1049.744,297.956,392.455,172.469,38.691,157.348
C04496=1049.751,298.204,392.424,172.473,38.694,157.349
C04497=1049.757,298.452,392.391,172.476,38.697,157.349
C04498=1049.764,298.699,392.359,172.479,38.701,157.350
C04499=1049.770,298.947,392.326,172.483,38.704,157.351
C04500=1049.776,299.195,392.293,172.487,38.707,157.352
C04501=1049.784,299.443,392.261,172.489,38.711,157.353
C04502=1049.790,299.690,392.228,172.493,38.714,157.354
C04503=1049.796,299.938,392.196,172.497,38.717,157.354
C04504=1049.803,300.186,392.163,172.500,38.720,157.355
C04505=1049.809,300.434,392.130,172.503,38.724,157.356
C04506=1049.816,300.682,392.098,172.507,38.727,157.357
C04507=1049.823,300.929,392.065,172.510,38.731,157.358
C04508=1049.829,301.177,392.032,172.513,38.734,157.358
C04509=1049.835,301.424,392.000,172.517,38.737,157.359
C04510=1049.842,301.673,391.966,172.520,38.741,157.360
C04511=1049.849,301.920,391.934,172.524,38.744,157.361
C04512=1049.856,302.167,391.902,172.527,38.747,157.362
C04513=1049.862,302.415,391.869,172.531,38.751,157.363
C04514=1049.869,302.663,391.836,172.534,38.754,157.363
C04515=1049.875,302.911,391.803,172.538,38.757,157.364
C04516=1049.881,303.159,391.770,172.541,38.761,157.365
C04517=1049.888,303.406,391.737,172.544,38.764,157.366
C04518=1049.895,303.654,391.705,172.548,38.768,157.367
C04519=1049.902,303.901,391.672,172.552,38.771,157.368
C04520=1049.908,304.149,391.639,172.555,38.774,157.368
C04521=1049.914,304.365,391.610,172.558,38.777,157.369
C04522=1049.920,304.581,391.582,172.561,38.780,157.370
C04523=1049.925,304.797,391.553,172.564,38.783,157.371
C04524=1049.931,305.013,391.524,172.567,38.786,157.371
C04525=1049.937,305.228,391.495,172.571,38.789,157.372
C04526=1049.943,305.444,391.466,172.573,38.792,157.373
C04527=1049.949,305.660,391.437,172.577,38.795,157.374
C04528=1049.954,305.876,391.409,172.580,38.798,157.374
C04529=1049.962,306.124,391.376,172.583,38.801,157.375
C04530=1049.968,306.371,391.344,172.587,38.804,157.376
C04531=1049.975,306.619,391.310,172.590,38.808,157.377
C04532=1049.982,306.866,391.277,172.594,38.811,157.378
C04533=1049.989,307.115,391.244,172.597,38.814,157.379
C04534=1049.995,307.362,391.210,172.601,38.818,157.379
C04535=1050.001,307.609,391.178,172.605,38.821,157.380
C04536=1050.008,307.858,391.145,172.608,38.825,157.381
C04537=1050.016,308.104,391.112,172.612,38.828,157.382
C04538=1050.023,308.353,391.079,172.615,38.832,157.383
C04539=1050.029,308.600,391.045,172.619,38.835,157.384
C04540=1050.036,308.848,391.012,172.623,38.838,157.385
C04541=1050.042,309.095,390.979,172.627,38.842,157.385
C04542=1050.050,309.343,390.946,172.629,38.845,157.386
C04543=1050.056,309.591,390.913,172.633,38.849,157.387
C04544=1050.063,309.838,390.879,172.637,38.852,157.388
C04545=1050.070,310.087,390.846,172.641,38.855,157.389
C04546=1050.076,310.334,390.812,172.645,38.859,157.390
C04547=1050.083,310.582,390.779,172.648,38.862,157.391
C04548=1050.091,310.829,390.746,172.652,38.866,157.391
C04549=1050.098,311.076,390.713,172.655,38.869,157.392
C04550=1050.104,311.324,390.680,172.659,38.872,157.393
C04551=1050.111,311.572,390.646,172.662,38.876,157.394
C04552=1050.118,311.820,390.613,172.666,38.879,157.395
C04553=1050.125,312.067,390.579,172.670,38.883,157.396
C04554=1050.132,312.314,390.546,172.674,38.886,157.397
C04555=1050.139,312.563,390.513,172.678,38.890,157.397
C04556=1050.146,312.810,390.479,172.681,38.893,157.398
C04557=1050.153,313.057,390.445,172.685,38.896,157.399
C04558=1050.158,313.305,390.412,172.689,38.900,157.400
C04559=1050.166,313.553,390.378,172.692,38.904,157.401
C04560=1050.172,313.801,390.344,172.696,38.908,157.402
C04561=1050.179,314.048,390.310,172.699,38.911,157.403
C04562=1050.186,314.296,390.276,172.703,38.915,157.404
C04563=1050.192,314.543,390.242,172.707,38.918,157.405
C04564=1050.199,314.791,390.209,172.711,38.922,157.406
C04565=1050.205,315.038,390.174,172.715,38.925,157.406
C04566=1050.212,315.286,390.141,172.719,38.929,157.407
C04567=1050.218,315.534,390.106,172.721,38.933,157.408
C04568=1050.225,315.780,390.073,172.725,38.936,157.409
C04569=1050.231,316.028,390.038,172.729,38.940,157.410
C04570=1050.239,316.276,390.005,172.733,38.944,157.411
C04571=1050.245,316.523,389.970,172.737,38.947,157.412
C04572=1050.252,316.771,389.937,172.741,38.951,157.413
C04573=1050.258,317.019,389.902,172.744,38.954,157.414
C04574=1050.265,317.266,389.869,172.748,38.958,157.415
C04575=1050.271,317.514,389.834,172.752,38.961,157.416
C04576=1050.278,317.762,389.801,172.756,38.965,157.417
C04577=1050.283,317.974,389.771,172.759,38.969,157.417
C04578=1050.290,318.187,389.741,172.762,38.971,157.418
C04579=1050.298,318.481,389.702,172.766,38.976,157.419
C04580=1050.305,318.777,389.660,172.771,38.980,157.420
C04581=1050.314,319.071,389.619,172.776,38.985,157.422
C04582=1050.321,319.366,389.579,172.781,38.989,157.423
C04583=1050.328,319.613,389.545,172.784,38.992,157.424
C04584=1050.335,319.861,389.510,172.788,38.996,157.425
C04585=1050.342,320.108,389.476,172.792,39.000,157.426
C04586=1050.348,320.356,389.442,172.796,39.004,157.426
C04587=1050.356,320.603,389.407,172.800,39.007,157.427
C04588=1050.362,320.851,389.373,172.804,39.011,157.428
C04589=1050.369,321.098,389.339,172.808,39.015,157.429
C04590=1050.376,321.346,389.304,172.811,39.019,157.430
C04591=1050.382,321.594,389.270,172.815,39.022,157.431
C04592=1050.389,321.841,389.236,172.819,39.026,157.432
C04593=1050.396,322.089,389.201,172.823,39.030,157.433
C04594=1050.403,322.336,389.167,172.827,39.033,157.434
C04595=1050.410,322.584,389.133,172.831,39.037,157.435
C04596=1050.417,322.831,389.098,172.835,39.041,157.436
C04597=1050.423,323.079,389.064,172.839,39.045,157.437
C04598=1050.430,323.326,389.029,172.842,39.048,157.438
C04599=1050.437,323.574,388.995,172.846,39.052,157.439
C04600=1050.444,323.821,388.960,172.850,39.056,157.440
C04601=1050.451,324.069,388.926,172.854,39.059,157.441
C04602=1050.458,324.316,388.891,172.858,39.063,157.442
C04603=1050.464,324.564,388.857,172.862,39.067,157.443
C04604=1050.472,324.811,388.822,172.867,39.070,157.444
C04605=1050.478,325.059,388.787,172.871,39.074,157.445
C04606=1050.486,325.306,388.753,172.875,39.078,157.446
C04607=1050.492,325.554,388.718,172.878,39.081,157.446
C04608=1050.499,325.802,388.684,172.882,39.085,157.447
C04609=1050.506,326.049,388.649,172.886,39.089,157.448
C04610=1050.513,326.296,388.614,172.890,39.093,157.449
C04611=1050.521,326.544,388.578,172.894,39.097,157.450
C04612=1050.528,326.792,388.545,172.898,39.101,157.451
C04613=1050.534,327.039,388.509,172.902,39.104,157.452
C04614=1050.542,327.286,388.475,172.907,39.108,157.453
C04615=1050.548,327.534,388.440,172.911,39.112,157.454
C04616=1050.555,327.781,388.405,172.915,39.116,157.455
C04617=1050.563,328.029,388.371,172.919,39.119,157.456
C04618=1050.570,328.276,388.336,172.922,39.123,157.457
C04619=1050.576,328.523,388.300,172.926,39.127,157.458
C04620=1050.584,328.772,388.266,172.931,39.131,157.459
C04621=1050.591,329.019,388.231,172.935,39.135,157.460
C04622=1050.598,329.266,388.196,172.939,39.139,157.461
C04623=1050.605,329.513,388.161,172.943,39.142,157.462
C04624=1050.612,329.761,388.126,172.947,39.146,157.463
C04625=1050.619,330.009,388.091,172.951,39.150,157.464
C04626=1050.626,330.256,388.056,172.956,39.154,157.465
C04627=1050.633,330.504,388.021,172.960,39.158,157.466
C04628=1050.640,330.751,387.985,172.964,39.162,157.467
C04629=1050.646,330.998,387.950,172.968,39.166,157.468
C04630=1050.653,331.246,387.915,172.972,39.169,157.469
C04631=1050.660,331.492,387.879,172.976,39.174,157.470
C04632=1050.668,331.740,387.844,172.981,39.178,157.471
C04633=1050.674,331.988,387.809,172.985,39.181,157.472
C04634=1050.681,332.235,387.774,172.989,39.185,157.473
C04635=1050.689,332.525,387.733,172.994,39.190,157.475
C04636=1050.697,332.814,387.690,172.998,39.195,157.476
C04637=1050.704,333.104,387.649,173.003,39.200,157.477
C04638=1050.713,333.394,387.607,173.008,39.204,157.478
C04639=1050.720,333.641,387.572,173.012,39.208,157.479
C04640=1050.727,333.889,387.537,173.016,39.212,157.480
C04641=1050.735,334.136,387.501,173.021,39.216,157.481
C04642=1050.741,334.383,387.465,173.025,39.220,157.482
C04643=1050.748,334.631,387.430,173.029,39.224,157.484
C04644=1050.755,334.877,387.394,173.033,39.228,157.485
C04645=1050.763,335.126,387.359,173.038,39.232,157.486
C04646=1050.770,335.372,387.323,173.042,39.236,157.487
C04647=1050.776,335.620,387.288,173.046,39.240,157.488
C04648=1050.783,335.868,387.252,173.050,39.244,157.489
C04649=1050.790,336.115,387.216,173.055,39.248,157.490
C04650=1050.797,336.363,387.181,173.059,39.252,157.491
C04651=1050.805,336.610,387.145,173.063,39.257,157.492
C04652=1050.812,336.856,387.109,173.068,39.260,157.493
C04653=1050.818,337.105,387.073,173.072,39.265,157.494
C04654=1050.825,337.351,387.037,173.076,39.269,157.495
C04655=1050.832,337.599,387.002,173.080,39.273,157.496
C04656=1050.839,337.847,386.965,173.085,39.277,157.497
C04657=1050.846,338.093,386.929,173.089,39.281,157.499
C04658=1050.853,338.341,386.894,173.093,39.286,157.500
C04659=1050.860,338.588,386.857,173.098,39.289,157.501
C04660=1050.867,338.835,386.821,173.102,39.294,157.502
C04661=1050.875,339.083,386.785,173.106,39.298,157.503
C04662=1050.881,339.330,386.749,173.112,39.302,157.504
C04663=1050.888,339.578,386.713,173.116,39.306,157.505
C04664=1050.895,339.824,386.677,173.120,39.310,157.506
C04665=1050.902,340.072,386.640,173.125,39.314,157.507
C04666=1050.909,340.319,386.605,173.129,39.319,157.508
C04667=1050.917,340.567,386.569,173.133,39.323,157.510
C04668=1050.923,340.814,386.533,173.138,39.327,157.511
C04669=1050.931,341.062,386.496,173.142,39.331,157.512
C04670=1050.937,341.309,386.460,173.146,39.336,157.513
C04671=1050.945,341.556,386.424,173.151,39.339,157.514
C04672=1050.952,341.803,386.388,173.155,39.344,157.515
C04673=1050.959,342.051,386.351,173.160,39.348,157.516
C04674=1050.966,342.297,386.315,173.164,39.353,157.517
C04675=1050.973,342.545,386.279,173.168,39.356,157.518
C04676=1050.980,342.792,386.243,173.173,39.361,157.520
C04677=1050.987,343.039,386.206,173.178,39.365,157.521
C04678=1050.994,343.287,386.170,173.182,39.369,157.522
C04679=1051.001,343.534,386.133,173.187,39.374,157.523
C04680=1051.008,343.781,386.097,173.191,39.378,157.524
C04681=1051.015,344.028,386.060,173.196,39.382,157.525
C04682=1051.023,344.275,386.024,173.200,39.387,157.527
C04683=1051.030,344.523,385.987,173.205,39.391,157.528
C04684=1051.036,344.770,385.950,173.209,39.396,157.529
C04685=1051.044,345.018,385.914,173.213,39.400,157.530
C04686=1051.050,345.264,385.877,173.219,39.404,157.531
C04687=1051.058,345.511,385.841,173.223,39.409,157.532
C04688=1051.065,345.759,385.804,173.228,39.413,157.534
C04689=1051.072,346.006,385.767,173.232,39.417,157.535
C04690=1051.079,346.253,385.731,173.237,39.422,157.536
C04691=1051.087,346.539,385.687,173.242,39.426,157.537
C04692=1051.096,346.825,385.646,173.248,39.432,157.539
C04693=1051.104,347.111,385.602,173.253,39.437,157.540
C04694=1051.112,347.395,385.560,173.258,39.442,157.541
C04695=1051.119,347.643,385.523,173.262,39.447,157.543
C04696=1051.127,347.890,385.486,173.268,39.451,157.544
C04697=1051.134,348.138,385.450,173.272,39.455,157.545
C04698=1051.140,348.384,385.413,173.277,39.460,157.546
C04699=1051.148,348.631,385.375,173.281,39.465,157.547
C04700=1051.155,348.879,385.339,173.286,39.469,157.548
C04701=1051.162,349.126,385.301,173.290,39.473,157.550
C04702=1051.169,349.373,385.265,173.295,39.477,157.551
C04703=1051.177,349.620,385.228,173.300,39.482,157.552
C04704=1051.184,349.867,385.190,173.305,39.487,157.553
C04705=1051.191,350.115,385.154,173.309,39.491,157.554
C04706=1051.198,350.362,385.116,173.314,39.496,157.556
C04707=1051.206,350.609,385.079,173.319,39.500,157.557
C04708=1051.213,350.856,385.042,173.324,39.505,157.558
C04709=1051.220,351.103,385.005,173.329,39.509,157.559
C04710=1051.227,351.350,384.968,173.333,39.514,157.561
C04711=1051.234,351.597,384.930,173.338,39.519,157.562
C04712=1051.241,351.844,384.893,173.342,39.523,157.563
C04713=1051.249,352.091,384.855,173.348,39.528,157.564
C04714=1051.256,352.339,384.817,173.352,39.533,157.566
C04715=1051.263,352.586,384.780,173.357,39.537,157.567
C04716=1051.270,352.833,384.742,173.362,39.542,157.568
C04717=1051.277,353.079,384.705,173.367,39.546,157.569
C04718=1051.284,353.326,384.668,173.372,39.551,157.571
C04719=1051.292,353.574,384.630,173.376,39.556,157.572
C04720=1051.299,353.821,384.593,173.381,39.560,157.573
C04721=1051.306,354.068,384.555,173.387,39.565,157.574
C04722=1051.313,354.315,384.518,173.391,39.569,157.576
C04723=1051.321,354.562,384.480,173.396,39.574,157.577
C04724=1051.328,354.809,384.443,173.401,39.579,157.578
C04725=1051.335,355.056,384.405,173.406,39.584,157.580
C04726=1051.342,355.304,384.368,173.411,39.588,157.581
C04727=1051.350,355.550,384.329,173.416,39.593,157.582
C04728=1051.357,355.797,384.292,173.420,39.598,157.583
C04729=1051.364,356.044,384.254,173.426,39.603,157.585
C04730=1051.372,356.291,384.217,173.431,39.607,157.586
C04731=1051.380,356.539,384.178,173.435,39.612,157.587
C04732=1051.387,356.786,384.141,173.440,39.617,157.589
C04733=1051.394,357.033,384.103,173.446,39.622,157.590
C04734=1051.402,357.279,384.065,173.450,39.627,157.591
C04735=1051.409,357.527,384.027,173.455,39.631,157.592
C04736=1051.416,357.774,383.990,173.461,39.636,157.594
C04737=1051.424,358.020,383.951,173.466,39.641,157.595
C04738=1051.431,358.267,383.914,173.470,39.646,157.596
C04739=1051.438,358.514,383.875,173.475,39.651,157.598
C04740=1051.446,358.762,383.837,173.481,39.656,157.599
C04741=1051.453,359.009,383.799,173.485,39.660,157.600
C04742=1051.460,359.256,383.761,173.490,39.665,157.602
C04743=1051.467,359.502,383.723,173.496,39.670,157.603
C04744=1051.475,359.749,383.684,173.501,39.675,157.604
C04745=1051.482,359.996,383.647,173.505,39.680,157.606
C04746=1051.490,360.243,383.608,173.511,39.685,157.607
C04747=1051.499,360.534,383.564,173.517,39.690,157.609
C04748=1051.507,360.825,383.518,173.523,39.696,157.610
C04749=1051.516,361.116,383.473,173.529,39.702,157.612
C04750=1051.525,361.407,383.428,173.535,39.708,157.614
C04751=1051.532,361.654,383.390,173.540,39.713,157.615
C04752=1051.539,361.901,383.351,173.546,39.718,157.616
C04753=1051.547,362.148,383.313,173.550,39.723,157.618
C04754=1051.555,362.394,383.274,173.555,39.728,157.619
C04755=1051.562,362.641,383.236,173.561,39.733,157.620
C04756=1051.569,362.888,383.197,173.566,39.738,157.622
C04757=1051.577,363.135,383.159,173.572,39.743,157.623
C04758=1051.584,363.382,383.120,173.577,39.748,157.625
C04759=1051.592,363.628,383.082,173.581,39.753,157.626
C04760=1051.599,363.876,383.042,173.587,39.759,157.627
C04761=1051.607,364.122,383.004,173.592,39.763,157.629
C04762=1051.613,364.369,382.965,173.598,39.769,157.630
C04763=1051.622,364.616,382.927,173.603,39.774,157.632
C04764=1051.628,364.863,382.888,173.609,39.779,157.633
C04765=1051.636,365.110,382.850,173.613,39.784,157.634
C04766=1051.643,365.357,382.810,173.618,39.790,157.636
C04767=1051.651,365.603,382.772,173.624,39.794,157.637
C04768=1051.659,365.851,382.732,173.629,39.800,157.639
C04769=1051.665,366.097,382.693,173.635,39.805,157.640
C04770=1051.674,366.345,382.655,173.640,39.810,157.642
C04771=1051.681,366.591,382.615,173.646,39.815,157.643
C04772=1051.688,366.837,382.577,173.651,39.821,157.645
C04773=1051.696,367.085,382.538,173.657,39.826,157.646
C04774=1051.704,367.331,382.499,173.662,39.831,157.648
C04775=1051.711,367.578,382.460,173.666,39.836,157.649
C04776=1051.718,367.824,382.420,173.672,39.841,157.650
C04777=1051.726,368.072,382.382,173.677,39.847,157.652
C04778=1051.733,368.318,382.342,173.683,39.852,157.653
C04779=1051.741,368.565,382.303,173.688,39.857,157.655
C04780=1051.749,368.812,382.263,173.694,39.863,157.656
C04781=1051.756,369.059,382.225,173.699,39.868,157.658
C04782=1051.764,369.305,382.185,173.705,39.873,157.659
C04783=1051.771,369.552,382.146,173.710,39.879,157.661
C04784=1051.780,369.799,382.107,173.716,39.884,157.662
C04785=1051.787,370.046,382.068,173.721,39.889,157.664
C04786=1051.794,370.293,382.028,173.727,39.895,157.665
C04787=1051.803,370.539,381.989,173.732,39.900,157.667
C04788=1051.810,370.785,381.949,173.738,39.905,157.668
C04789=1051.817,371.033,381.910,173.744,39.911,157.670
C04790=1051.826,371.279,381.871,173.749,39.917,157.671
C04791=1051.833,371.526,381.831,173.755,39.922,157.673
C04792=1051.841,371.773,381.791,173.761,39.927,157.674
C04793=1051.848,372.019,381.752,173.767,39.932,157.676
C04794=1051.856,372.267,381.713,173.772,39.938,157.677
C04795=1051.864,372.513,381.673,173.778,39.944,157.679
C04796=1051.871,372.760,381.633,173.784,39.949,157.681
C04797=1051.879,373.007,381.594,173.789,39.955,157.682
C04798=1051.886,373.253,381.554,173.795,39.961,157.684
C04799=1051.894,373.500,381.514,173.800,39.966,157.685
C04800=1051.902,373.746,381.473,173.806,39.972,157.687
C04801=1051.909,373.992,381.434,173.812,39.977,157.688
C04802=1051.917,374.239,381.394,173.817,39.983,157.690
C04803=1051.927,374.549,381.344,173.824,39.990,157.692
C04804=1051.936,374.859,381.293,173.832,39.997,157.694
C04805=1051.946,375.169,381.244,173.839,40.004,157.696
C04806=1051.956,375.478,381.193,173.846,40.011,157.698
C04807=1051.963,375.725,381.153,173.852,40.017,157.700
C04808=1051.971,375.972,381.113,173.858,40.022,157.701
C04809=1051.979,376.219,381.073,173.863,40.028,157.703
C04810=1051.986,376.465,381.033,173.870,40.034,157.704
C04811=1051.994,376.712,380.993,173.876,40.040,157.706
C04812=1052.002,376.958,380.953,173.881,40.045,157.708
C04813=1052.010,377.205,380.913,173.887,40.051,157.709
C04814=1052.018,377.451,380.872,173.893,40.057,157.711
C04815=1052.025,377.698,380.832,173.899,40.062,157.712
C04816=1052.033,377.944,380.791,173.905,40.068,157.714
C04817=1052.041,378.191,380.752,173.911,40.074,157.716
C04818=1052.049,378.438,380.711,173.916,40.080,157.717
C04819=1052.057,378.684,380.671,173.922,40.086,157.719
C04820=1052.065,378.931,380.630,173.929,40.091,157.721
C04821=1052.073,379.177,380.590,173.935,40.097,157.722
C04822=1052.081,379.424,380.550,173.940,40.103,157.724
C04823=1052.089,379.670,380.509,173.947,40.109,157.726
C04824=1052.097,379.916,380.469,173.953,40.115,157.727
C04825=1052.104,380.163,380.429,173.959,40.121,157.729
C04826=1052.112,380.410,380.388,173.964,40.127,157.731
C04827=1052.120,380.656,380.347,173.971,40.133,157.732
C04828=1052.128,380.903,380.306,173.977,40.139,157.734
C04829=1052.136,381.150,380.265,173.983,40.145,157.736
C04830=1052.144,381.396,380.224,173.988,40.151,157.738
C04831=1052.152,381.642,380.183,173.995,40.157,157.739
C04832=1052.160,381.889,380.143,174.001,40.163,157.741
C04833=1052.167,382.135,380.101,174.007,40.169,157.743
C04834=1052.175,382.382,380.061,174.014,40.175,157.745
C04835=1052.183,382.628,380.020,174.019,40.181,157.746
C04836=1052.190,382.874,379.979,174.025,40.187,157.748
C04837=1052.199,383.121,379.938,174.032,40.193,157.750
C04838=1052.207,383.368,379.897,174.038,40.200,157.752
C04839=1052.215,383.614,379.855,174.045,40.205,157.753
C04840=1052.223,383.860,379.815,174.051,40.212,157.755
C04841=1052.231,384.106,379.774,174.056,40.218,157.757
C04842=1052.239,384.354,379.732,174.063,40.224,157.759
C04843=1052.247,384.599,379.691,174.069,40.230,157.760
C04844=1052.255,384.845,379.650,174.076,40.236,157.762
C04845=1052.262,385.092,379.609,174.082,40.243,157.764
C04846=1052.271,385.338,379.568,174.088,40.249,157.766
C04847=1052.278,385.585,379.526,174.095,40.255,157.768
C04848=1052.286,385.831,379.486,174.101,40.262,157.770
C04849=1052.295,386.078,379.444,174.107,40.267,157.771
C04850=1052.303,386.324,379.403,174.113,40.274,157.773
C04851=1052.311,386.570,379.361,174.120,40.280,157.775
C04852=1052.319,386.817,379.320,174.126,40.286,157.777
C04853=1052.327,387.063,379.278,174.133,40.293,157.779
C04854=1052.336,387.309,379.237,174.139,40.299,157.780
C04855=1052.343,387.556,379.195,174.146,40.305,157.782
C04856=1052.352,387.802,379.154,174.152,40.312,157.784
C04857=1052.360,388.048,379.112,174.159,40.318,157.786
C04858=1052.369,388.295,379.071,174.165,40.324,157.788
C04859=1052.380,388.636,379.013,174.175,40.333,157.790
C04860=1052.392,388.979,378.955,174.183,40.342,157.793
C04861=1052.403,389.321,378.897,174.192,40.351,157.796
C04862=1052.414,389.663,378.839,174.202,40.360,157.798
C04863=1052.422,389.909,378.797,174.208,40.367,157.800
C04864=1052.431,390.156,378.756,174.215,40.373,157.802
C04865=1052.439,390.402,378.713,174.221,40.380,157.804
C04866=1052.446,390.648,378.672,174.228,40.387,157.806
C04867=1052.456,390.894,378.629,174.235,40.393,157.808
C04868=1052.463,391.140,378.587,174.241,40.400,157.810
C04869=1052.471,391.387,378.545,174.248,40.406,157.812
C04870=1052.480,391.633,378.503,174.255,40.413,157.814
C04871=1052.488,391.879,378.461,174.261,40.419,157.816
C04872=1052.496,392.126,378.419,174.268,40.426,157.818
C04873=1052.505,392.372,378.376,174.276,40.433,157.820
C04874=1052.513,392.618,378.334,174.282,40.440,157.822
C04875=1052.521,392.864,378.292,174.289,40.447,157.824
C04876=1052.530,393.110,378.249,174.296,40.453,157.826
C04877=1052.537,393.356,378.207,174.302,40.460,157.827
C04878=1052.546,393.603,378.165,174.309,40.467,157.829
C04879=1052.555,393.849,378.122,174.316,40.474,157.831
C04880=1052.562,394.095,378.080,174.324,40.480,157.833
C04881=1052.571,394.341,378.037,174.330,40.487,157.835
C04882=1052.579,394.587,377.995,174.337,40.494,157.838
C04883=1052.588,394.833,377.952,174.344,40.501,157.840
C04884=1052.596,395.079,377.909,174.351,40.508,157.842
C04885=1052.604,395.325,377.867,174.357,40.515,157.844
C04886=1052.613,395.571,377.825,174.365,40.522,157.846
C04887=1052.621,395.817,377.782,174.372,40.529,157.848
C04888=1052.630,396.064,377.739,174.379,40.535,157.850
C04889=1052.638,396.310,377.696,174.386,40.543,157.852
C04890=1052.647,396.556,377.653,174.393,40.549,157.854
C04891=1052.655,396.802,377.610,174.400,40.557,157.856
C04892=1052.664,397.048,377.567,174.407,40.563,157.858
C04893=1052.672,397.295,377.525,174.414,40.571,157.860
C04894=1052.680,397.541,377.482,174.422,40.578,157.862
C04895=1052.689,397.787,377.439,174.429,40.585,157.864
C04896=1052.697,398.033,377.396,174.435,40.592,157.867
C04897=1052.706,398.279,377.353,174.443,40.599,157.869
C04898=1052.714,398.525,377.310,174.450,40.606,157.871
C04899=1052.723,398.771,377.266,174.457,40.614,157.873
C04900=1052.731,399.017,377.222,174.465,40.621,157.875
C04901=1052.739,399.263,377.179,174.472,40.628,157.877
C04902=1052.748,399.509,377.136,174.479,40.635,157.879
C04903=1052.756,399.755,377.093,174.486,40.642,157.882
C04904=1052.765,400.001,377.050,174.494,40.649,157.884
C04905=1052.774,400.247,377.007,174.501,40.657,157.886
C04906=1052.782,400.493,376.964,174.509,40.664,157.888
C04907=1052.791,400.739,376.920,174.516,40.672,157.890
C04908=1052.800,400.985,376.876,174.523,40.679,157.893
C04909=1052.808,401.231,376.833,174.531,40.686,157.895
C04910=1052.816,401.477,376.790,174.538,40.694,157.897
C04911=1052.826,401.723,376.746,174.546,40.701,157.899
C04912=1052.834,401.969,376.703,174.553,40.708,157.901
C04913=1052.842,402.215,376.658,174.561,40.716,157.904
C04914=1052.852,402.461,376.614,174.568,40.723,157.906
C04915=1052.864,402.821,376.551,174.579,40.734,157.909
C04916=1052.877,403.182,376.486,174.590,40.745,157.913
C04917=1052.890,403.542,376.423,174.601,40.756,157.916
C04918=1052.903,403.902,376.358,174.612,40.767,157.919
C04919=1052.911,404.148,376.314,174.620,40.775,157.922
C04920=1052.920,404.395,376.270,174.628,40.783,157.924
C04921=1052.928,404.640,376.226,174.635,40.790,157.926
C04922=1052.937,404.887,376.182,174.643,40.798,157.928
C04923=1052.946,405.132,376.138,174.650,40.805,157.931
C04924=1052.954,405.378,376.093,174.658,40.813,157.933
C04925=1052.963,405.624,376.049,174.667,40.821,157.936
C04926=1052.972,405.870,376.005,174.674,40.829,157.938
C04927=1052.981,406.115,375.960,174.682,40.837,157.940
C04928=1052.989,406.361,375.916,174.690,40.844,157.943
C04929=1052.998,406.607,375.871,174.697,40.852,157.945
C04930=1053.007,406.853,375.827,174.706,40.860,157.948
C04931=1053.015,407.099,375.783,174.713,40.868,157.950
C04932=1053.025,407.345,375.738,174.721,40.876,157.952
C04933=1053.033,407.590,375.694,174.729,40.884,157.955
C04934=1053.043,407.837,375.649,174.737,40.892,157.957
C04935=1053.052,408.082,375.604,174.745,40.900,157.960
C04936=1053.060,408.328,375.560,174.753,40.908,157.962
C04937=1053.069,408.574,375.515,174.762,40.916,157.964
C04938=1053.078,408.820,375.470,174.769,40.924,157.967
C04939=1053.087,409.065,375.426,174.777,40.932,157.969
C04940=1053.096,409.311,375.381,174.786,40.940,157.972
C04941=1053.105,409.557,375.336,174.794,40.948,157.974
C04942=1053.114,409.803,375.291,174.802,40.956,157.977
C04943=1053.123,410.049,375.246,174.810,40.964,157.979
C04944=1053.132,410.294,375.201,174.818,40.972,157.982
C04945=1053.141,410.540,375.156,174.827,40.980,157.984
C04946=1053.150,410.786,375.111,174.835,40.989,157.987
C04947=1053.160,411.032,375.067,174.844,40.997,157.989
C04948=1053.169,411.278,375.021,174.851,41.005,157.992
C04949=1053.178,411.523,374.976,174.860,41.013,157.995
C04950=1053.187,411.769,374.931,174.868,41.022,157.997
C04951=1053.196,412.015,374.886,174.877,41.030,158.000
C04952=1053.205,412.261,374.840,174.885,41.038,158.002
C04953=1053.215,412.506,374.795,174.894,41.047,158.005
C04954=1053.224,412.752,374.750,174.902,41.055,158.007
C04955=1053.233,412.998,374.704,174.911,41.063,158.010
C04956=1053.242,413.244,374.659,174.919,41.072,158.013
C04957=1053.252,413.489,374.614,174.928,41.080,158.015
C04958=1053.261,413.735,374.569,174.937,41.088,158.018
C04959=1053.270,413.980,374.523,174.945,41.097,158.021
C04960=1053.279,414.226,374.477,174.954,41.105,158.023
C04961=1053.288,414.472,374.432,174.962,41.114,158.026
C04962=1053.298,414.718,374.385,174.971,41.123,158.029
C04963=1053.307,414.963,374.340,174.980,41.131,158.031
C04964=1053.316,415.209,374.294,174.988,41.140,158.034
C04965=1053.325,415.454,374.248,174.997,41.149,158.037
C04966=1053.334,415.700,374.202,175.006,41.157,158.039
C04967=1053.344,415.945,374.156,175.015,41.166,158.042
C04968=1053.353,416.191,374.110,175.023,41.175,158.045
C04969=1053.362,416.437,374.064,175.032,41.183,158.048
C04970=1053.372,416.682,374.018,175.041,41.192,158.050
C04971=1053.385,417.049,373.949,175.054,41.205,158.055
C04972=1053.399,417.415,373.880,175.068,41.218,158.059
C04973=1053.414,417.782,373.811,175.082,41.232,158.063
C04974=1053.428,418.148,373.743,175.096,41.245,158.067
C04975=1053.438,418.394,373.697,175.105,41.254,158.070
C04976=1053.447,418.639,373.650,175.113,41.263,158.073
C04977=1053.457,418.885,373.604,175.122,41.272,158.076
C04978=1053.466,419.130,373.557,175.132,41.281,158.079
C04979=1053.476,419.376,373.510,175.141,41.290,158.081
C04980=1053.485,419.621,373.464,175.150,41.299,158.084
C04981=1053.495,419.867,373.417,175.159,41.308,158.087
C04982=1053.504,420.111,373.371,175.169,41.317,158.090
C04983=1053.514,420.358,373.323,175.178,41.327,158.093
C04984=1053.523,420.603,373.277,175.188,41.336,158.096
C04985=1053.533,420.848,373.230,175.197,41.345,158.099
C04986=1053.542,421.094,373.183,175.206,41.354,158.102
C04987=1053.552,421.339,373.136,175.216,41.363,158.105
C04988=1053.562,421.585,373.090,175.225,41.373,158.108
C04989=1053.571,421.830,373.042,175.235,41.382,158.111
C04990=1053.581,422.075,372.995,175.244,41.391,158.114
C04991=1053.591,422.321,372.948,175.255,41.401,158.117
C04992=1053.600,422.565,372.902,175.264,41.410,158.120
C04993=1053.610,422.811,372.854,175.274,41.419,158.123
C04994=1053.620,423.056,372.807,175.283,41.429,158.126
C04995=1053.629,423.302,372.759,175.293,41.438,158.129
C04996=1053.639,423.547,372.713,175.303,41.448,158.132
C04997=1053.649,423.792,372.665,175.313,41.457,158.135
C04998=1053.658,424.038,372.618,175.323,41.467,158.138
C04999=1053.668,424.283,372.570,175.332,41.477,158.141
C05000=1053.679,424.528,372.522,175.343,41.486,158.144
C05001=1053.688,424.774,372.475,175.352,41.496,158.148
C05002=1053.699,425.019,372.427,175.362,41.506,158.151
C05003=1053.709,425.264,372.380,175.373,41.515,158.154
C05004=1053.718,425.510,372.332,175.382,41.525,158.157
C05005=1053.728,425.755,372.285,175.392,41.534,158.160
C05006=1053.738,426.000,372.237,175.403,41.544,158.163
C05007=1053.748,426.245,372.189,175.413,41.554,158.167
C05008=1053.758,426.490,372.141,175.422,41.564,158.170
C05009=1053.768,426.736,372.093,175.433,41.574,158.173
C05010=1053.778,426.981,372.045,175.443,41.584,158.176
C05011=1053.788,427.226,371.997,175.454,41.593,158.179
C05012=1053.798,427.471,371.949,175.464,41.604,158.183
C05013=1053.808,427.716,371.901,175.474,41.614,158.186
C05014=1053.817,427.961,371.853,175.484,41.624,158.189
C05015=1053.828,428.207,371.805,175.495,41.634,158.193
C05016=1053.838,428.452,371.756,175.505,41.644,158.196
C05017=1053.849,428.696,371.708,175.516,41.654,158.199
C05018=1053.858,428.941,371.660,175.527,41.664,158.203
C05019=1053.869,429.187,371.611,175.537,41.674,158.206
C05020=1053.879,429.432,371.563,175.548,41.685,158.209
C05021=1053.889,429.677,371.514,175.559,41.694,158.213
C05022=1053.899,429.922,371.466,175.569,41.705,158.216
C05023=1053.909,430.167,371.417,175.580,41.715,158.220
C05024=1053.919,430.412,371.369,175.591,41.725,158.223
C05025=1053.930,430.658,371.320,175.601,41.736,158.226
C05026=1053.940,430.902,371.271,175.612,41.746,158.230
C05027=1053.954,431.244,371.202,175.628,41.761,158.235
C05028=1053.968,431.585,371.135,175.643,41.776,158.240
C05029=1053.982,431.927,371.067,175.659,41.790,158.245
C05030=1053.997,432.269,370.998,175.673,41.805,158.250
C05031=1054.007,432.514,370.948,175.684,41.816,158.253
C05032=1054.017,432.758,370.899,175.696,41.826,158.257
C05033=1054.028,433.003,370.850,175.707,41.837,158.260
C05034=1054.039,433.248,370.802,175.718,41.847,158.264
C05035=1054.049,433.493,370.752,175.730,41.858,158.267
C05036=1054.060,433.738,370.702,175.741,41.869,158.271
C05037=1054.070,433.982,370.653,175.752,41.880,158.275
C05038=1054.081,434.227,370.604,175.764,41.891,158.278
C05039=1054.091,434.473,370.554,175.775,41.902,158.282
C05040=1054.101,434.717,370.505,175.786,41.912,158.286
C05041=1054.112,434.962,370.455,175.798,41.923,158.289
C05042=1054.123,435.207,370.406,175.809,41.934,158.293
C05043=1054.134,435.451,370.355,175.821,41.945,158.297
C05044=1054.144,435.696,370.306,175.833,41.956,158.301
C05045=1054.155,435.942,370.256,175.845,41.967,158.304
C05046=1054.165,436.185,370.206,175.856,41.978,158.308
C05047=1054.176,436.430,370.156,175.868,41.989,158.312
C05048=1054.187,436.675,370.107,175.880,42.001,158.316
C05049=1054.198,436.921,370.056,175.892,42.012,158.320
C05050=1054.208,437.165,370.007,175.904,42.023,158.323
C05051=1054.219,437.409,369.957,175.915,42.034,158.327
C05052=1054.230,437.654,369.906,175.928,42.045,158.331
C05053=1054.241,437.898,369.856,175.940,42.057,158.335
C05054=1054.253,438.144,369.806,175.951,42.068,158.339
C05055=1054.263,438.389,369.755,175.964,42.080,158.343
C05056=1054.274,438.633,369.705,175.976,42.091,158.347
C05057=1054.285,438.878,369.654,175.989,42.102,158.351
C05058=1054.296,439.122,369.604,176.001,42.114,158.355
C05059=1054.309,439.414,369.544,176.015,42.128,158.359
C05060=1054.322,439.705,369.483,176.030,42.142,158.364
C05061=1054.335,439.997,369.423,176.045,42.156,158.369
C05062=1054.348,440.288,369.361,176.060,42.170,158.374
C05063=1054.359,440.532,369.311,176.073,42.181,158.378
C05064=1054.370,440.777,369.260,176.085,42.193,158.382
C05065=1054.382,441.021,369.209,176.098,42.205,158.386
C05066=1054.393,441.267,369.158,176.111,42.216,158.390
C05067=1054.404,441.510,369.107,176.124,42.228,158.394
C05068=1054.415,441.754,369.056,176.136,42.241,158.399
C05069=1054.426,442.000,369.005,176.149,42.253,158.403
C05070=1054.437,442.244,368.954,176.163,42.264,158.407
C05071=1054.449,442.488,368.902,176.176,42.276,158.411
C05072=1054.460,442.732,368.851,176.189,42.288,158.415
C05073=1054.471,442.977,368.799,176.201,42.301,158.420
C05074=1054.482,443.221,368.748,176.214,42.312,158.424
C05075=1054.494,443.465,368.696,176.228,42.325,158.428
C05076=1054.505,443.710,368.644,176.241,42.337,158.432
C05077=1054.516,443.954,368.593,176.254,42.349,158.437
C05078=1054.527,444.199,368.541,176.268,42.362,158.441
C05079=1054.539,444.443,368.490,176.281,42.374,158.446
C05080=1054.550,444.687,368.437,176.294,42.386,158.450
C05081=1054.562,444.931,368.386,176.308,42.398,158.454
C05082=1054.573,445.176,368.334,176.322,42.411,158.459
C05083=1054.587,445.459,368.273,176.338,42.426,158.464
C05084=1054.601,445.743,368.214,176.354,42.440,158.469
C05085=1054.614,446.026,368.153,176.370,42.455,158.474
C05086=1054.628,446.309,368.092,176.386,42.469,158.480
C05087=1054.639,446.552,368.041,176.400,42.482,158.484
C05088=1054.651,446.795,367.989,176.413,42.494,158.489
C05089=1054.665,447.039,367.938,176.428,42.507,158.493
C05090=1054.679,447.283,367.887,176.441,42.518,158.497
C05091=1054.693,447.527,367.837,176.456,42.530,158.502
C05092=1054.709,447.771,367.788,176.470,42.542,158.506
C05093=1054.725,448.014,367.739,176.484,42.554,158.510
C05094=1054.742,448.259,367.691,176.499,42.565,158.515
C05095=1054.759,448.504,367.644,176.514,42.576,158.519
C05096=1054.778,448.749,367.597,176.528,42.587,158.523
C05097=1054.798,448.993,367.549,176.543,42.598,158.527
C05098=1054.817,449.238,367.504,176.557,42.609,158.531
C05099=1054.839,449.483,367.459,176.572,42.619,158.535
C05100=1054.860,449.729,367.413,176.587,42.629,158.539
C05101=1054.883,449.974,367.369,176.602,42.640,158.543
C05102=1054.906,450.220,367.326,176.617,42.649,158.547
C05103=1054.585,450.239,367.035,176.616,42.751,158.576
C05104=1054.561,449.994,367.079,176.600,42.741,158.572
C05105=1054.539,449.748,367.122,176.585,42.731,158.568
C05106=1054.517,449.503,367.167,176.570,42.721,158.564
C05107=1054.496,449.258,367.213,176.555,42.710,158.560
C05108=1054.476,449.013,367.259,176.541,42.700,158.556
C05109=1054.456,448.768,367.305,176.526,42.689,158.552
C05110=1054.438,448.523,367.353,176.510,42.678,158.547
C05111=1054.420,448.279,367.400,176.496,42.667,158.543
C05112=1054.402,448.035,367.448,176.482,42.655,158.539
C05113=1054.386,447.790,367.497,176.467,42.644,158.535
C05114=1054.370,447.546,367.546,176.453,42.632,158.530
C05115=1054.355,447.303,367.595,176.439,42.621,158.526
C05116=1054.341,447.059,367.646,176.424,42.609,158.522
C05117=1054.328,446.815,367.697,176.411,42.596,158.517
C05118=1054.315,446.571,367.748,176.396,42.584,158.513
C05119=1054.303,446.329,367.801,176.382,42.572,158.508
C05120=1054.291,446.064,367.857,176.367,42.558,158.503
C05121=1054.278,445.799,367.913,176.352,42.545,158.498
C05122=1054.265,445.536,367.970,176.337,42.531,158.493
C05123=1054.252,445.271,368.026,176.322,42.518,158.489
C05124=1054.241,445.026,368.078,176.309,42.505,158.484
C05125=1054.230,444.783,368.130,176.295,42.493,158.480
C05126=1054.219,444.538,368.182,176.282,42.481,158.475
C05127=1054.206,444.294,368.234,176.268,42.468,158.471
C05128=1054.195,444.050,368.286,176.255,42.456,158.467
C05129=1054.184,443.805,368.337,176.241,42.444,158.462
C05130=1054.172,443.561,368.389,176.228,42.432,158.458
C05131=1054.161,443.316,368.441,176.215,42.420,158.454
C05132=1054.150,443.072,368.492,176.201,42.408,158.449
C05133=1054.139,442.827,368.544,176.188,42.396,158.445
C05134=1054.127,442.584,368.595,176.175,42.384,158.441
C05135=1054.116,442.339,368.647,176.162,42.372,158.437
C05136=1054.105,442.095,368.698,176.149,42.360,158.432
C05137=1054.093,441.850,368.749,176.135,42.348,158.428
C05138=1054.082,441.606,368.801,176.122,42.336,158.424
C05139=1054.071,441.361,368.851,176.110,42.324,158.420
C05140=1054.059,441.117,368.903,176.097,42.312,158.416
C05141=1054.049,440.872,368.954,176.084,42.300,158.412
C05142=1054.037,440.628,369.005,176.072,42.289,158.408
C05143=1054.026,440.383,369.056,176.059,42.277,158.403
C05144=1054.015,440.139,369.107,176.046,42.266,158.399
C05145=1054.004,439.894,369.157,176.034,42.254,158.395
C05146=1053.993,439.650,369.208,176.021,42.243,158.391
C05147=1053.982,439.405,369.259,176.008,42.231,158.387
C05148=1053.971,439.161,369.310,175.996,42.219,158.383
C05149=1053.960,438.916,369.360,175.983,42.208,158.379
C05150=1053.949,438.672,369.411,175.971,42.196,158.375
C05151=1053.938,438.428,369.461,175.959,42.185,158.371
C05152=1053.927,438.182,369.512,175.947,42.173,158.367
C05153=1053.916,437.937,369.561,175.935,42.162,158.364
C05154=1053.906,437.693,369.612,175.922,42.151,158.360
C05155=1053.895,437.448,369.663,175.910,42.140,158.356
C05156=1053.884,437.204,369.713,175.898,42.129,158.352
C05157=1053.873,436.959,369.763,175.886,42.117,158.348
C05158=1053.862,436.714,369.813,175.874,42.106,158.344
C05159=1053.851,436.470,369.863,175.863,42.095,158.340
C05160=1053.841,436.225,369.913,175.850,42.084,158.337
C05161=1053.830,435.980,369.962,175.839,42.073,158.333
C05162=1053.819,435.735,370.013,175.827,42.062,158.329
C05163=1053.808,435.490,370.062,175.816,42.051,158.325
C05164=1053.798,435.245,370.112,175.803,42.040,158.321
C05165=1053.787,435.001,370.162,175.792,42.029,158.318
C05166=1053.777,434.756,370.212,175.780,42.019,158.314
C05167=1053.765,434.512,370.261,175.769,42.008,158.310
C05168=1053.755,434.267,370.310,175.757,41.997,158.307
C05169=1053.744,434.022,370.359,175.746,41.986,158.303
C05170=1053.734,433.777,370.409,175.734,41.975,158.299
C05171=1053.723,433.532,370.459,175.723,41.964,158.296
C05172=1053.712,433.287,370.508,175.712,41.954,158.292
C05173=1053.702,433.043,370.557,175.700,41.943,158.289
C05174=1053.692,432.798,370.607,175.689,41.933,158.285
C05175=1053.682,432.553,370.656,175.678,41.922,158.281
C05176=1053.671,432.306,370.705,175.666,41.912,158.278
C05177=1053.661,432.060,370.755,175.655,41.901,158.274
C05178=1053.650,431.813,370.804,175.644,41.891,158.271
C05179=1053.640,431.567,370.854,175.633,41.880,158.267
C05180=1053.628,431.279,370.911,175.620,41.867,158.263
C05181=1053.616,430.990,370.969,175.607,41.855,158.259
C05182=1053.605,430.745,371.017,175.596,41.845,158.255
C05183=1053.595,430.500,371.067,175.586,41.834,158.252
C05184=1053.585,430.255,371.115,175.574,41.824,158.249
C05185=1053.575,430.010,371.164,175.563,41.814,158.245
C05186=1053.565,429.765,371.213,175.552,41.803,158.242
C05187=1053.555,429.520,371.261,175.542,41.794,158.238
C05188=1053.544,429.274,371.309,175.531,41.783,158.235
C05189=1053.534,429.029,371.358,175.520,41.773,158.232
C05190=1053.524,428.785,371.406,175.510,41.763,158.228
C05191=1053.514,428.540,371.454,175.499,41.753,158.225
C05192=1053.503,428.294,371.503,175.488,41.743,158.221
C05193=1053.493,428.049,371.551,175.478,41.733,158.218
C05194=1053.483,427.804,371.600,175.468,41.723,158.215
C05195=1053.473,427.559,371.648,175.458,41.713,158.212
C05196=1053.463,427.314,371.696,175.447,41.703,158.208
C05197=1053.453,427.068,371.744,175.437,41.693,158.205
C05198=1053.442,426.824,371.792,175.426,41.683,158.202
C05199=1053.433,426.578,371.840,175.416,41.673,158.199
C05200=1053.422,426.333,371.888,175.405,41.664,158.195
C05201=1053.413,426.088,371.936,175.396,41.654,158.192
C05202=1053.403,425.843,371.984,175.386,41.644,158.189
C05203=1053.393,425.598,372.032,175.375,41.634,158.186
C05204=1053.384,425.352,372.079,175.365,41.625,158.183
C05205=1053.373,425.107,372.127,175.355,41.615,158.179
C05206=1053.363,424.862,372.175,175.345,41.606,158.176
C05207=1053.353,424.616,372.222,175.335,41.596,158.173
C05208=1053.343,424.371,372.270,175.325,41.586,158.170
C05209=1053.333,424.126,372.317,175.315,41.577,158.167
C05210=1053.324,423.880,372.365,175.305,41.567,158.164
C05211=1053.314,423.636,372.412,175.295,41.558,158.161
C05212=1053.304,423.390,372.459,175.285,41.548,158.158
C05213=1053.294,423.145,372.507,175.276,41.539,158.154
C05214=1053.284,422.900,372.554,175.266,41.529,158.151
C05215=1053.274,422.654,372.601,175.256,41.520,158.148
C05216=1053.265,422.409,372.648,175.246,41.511,158.145
C05217=1053.255,422.163,372.695,175.236,41.501,158.142
C05218=1053.245,421.918,372.742,175.227,41.492,158.139
C05219=1053.236,421.673,372.790,175.217,41.483,158.136
C05220=1053.226,421.427,372.836,175.208,41.473,158.133
C05221=1053.216,421.182,372.883,175.198,41.464,158.130
C05222=1053.208,420.937,372.930,175.189,41.455,158.127
C05223=1053.197,420.691,372.977,175.180,41.446,158.124
C05224=1053.188,420.445,373.024,175.170,41.437,158.122
C05225=1053.179,420.201,373.071,175.161,41.428,158.119
C05226=1053.169,419.955,373.118,175.151,41.418,158.116
C05227=1053.160,419.709,373.164,175.142,41.409,158.113
C05228=1053.149,419.464,373.211,175.133,41.400,158.110
C05229=1053.140,419.219,373.257,175.123,41.391,158.107
C05230=1053.130,418.973,373.304,175.114,41.382,158.104
C05231=1053.121,418.728,373.350,175.105,41.374,158.101
C05232=1053.112,418.482,373.397,175.095,41.365,158.098
C05233=1053.102,418.236,373.443,175.086,41.355,158.095
C05234=1053.088,417.868,373.513,175.072,41.342,158.091
C05235=1053.073,417.499,373.582,175.058,41.329,158.087
C05236=1053.059,417.131,373.652,175.046,41.316,158.083
C05237=1053.045,416.762,373.720,175.032,41.303,158.079
C05238=1053.035,416.517,373.767,175.023,41.294,158.076
C05239=1053.026,416.271,373.813,175.013,41.286,158.073
C05240=1053.017,416.026,373.859,175.004,41.276,158.070
C05241=1053.008,415.780,373.904,174.996,41.268,158.068
C05242=1052.998,415.534,373.951,174.987,41.259,158.065
C05243=1052.989,415.289,373.997,174.978,41.251,158.062
C05244=1052.980,415.043,374.042,174.970,41.242,158.059
C05245=1052.970,414.798,374.089,174.961,41.233,158.057
C05246=1052.961,414.552,374.134,174.952,41.225,158.054
C05247=1052.952,414.307,374.180,174.944,41.216,158.051
C05248=1052.943,414.061,374.226,174.935,41.208,158.049
C05249=1052.934,413.815,374.271,174.926,41.200,158.046
C05250=1052.924,413.570,374.317,174.917,41.191,158.043
C05251=1052.915,413.324,374.363,174.908,41.182,158.041
C05252=1052.906,413.078,374.408,174.899,41.174,158.038
C05253=1052.897,412.832,374.453,174.892,41.166,158.036
C05254=1052.888,412.587,374.499,174.883,41.157,158.033
C05255=1052.878,412.341,374.543,174.875,41.149,158.030
C05256=1052.869,412.095,374.589,174.866,41.141,158.028
C05257=1052.860,411.849,374.634,174.858,41.133,158.025
C05258=1052.850,411.604,374.679,174.849,41.124,158.023
C05259=1052.841,411.358,374.724,174.841,41.116,158.020
C05260=1052.832,411.112,374.770,174.832,41.108,158.017
C05261=1052.823,410.867,374.815,174.824,41.100,158.015
C05262=1052.814,410.621,374.860,174.815,41.092,158.012
C05263=1052.805,410.375,374.906,174.808,41.084,158.010
C05264=1052.795,410.129,374.950,174.799,41.076,158.007
C05265=1052.787,409.884,374.995,174.791,41.067,158.005
C05266=1052.778,409.638,375.040,174.782,41.059,158.002
C05267=1052.768,409.392,375.084,174.774,41.051,158.000
C05268=1052.759,409.146,375.130,174.766,41.044,157.997
C05269=1052.750,408.901,375.174,174.758,41.035,157.995
C05270=1052.742,408.655,375.219,174.750,41.027,157.992
C05271=1052.733,408.409,375.264,174.741,41.020,157.990
C05272=1052.723,408.163,375.308,174.733,41.011,157.987
C05273=1052.715,407.918,375.353,174.726,41.004,157.985
C05274=1052.706,407.672,375.398,174.717,40.996,157.983
C05275=1052.697,407.425,375.442,174.709,40.988,157.980
C05276=1052.688,407.180,375.487,174.701,40.980,157.978
C05277=1052.679,406.934,375.531,174.694,40.972,157.975
C05278=1052.670,406.687,375.576,174.685,40.964,157.973
C05279=1052.662,406.442,375.620,174.677,40.957,157.971
C05280=1052.653,406.196,375.665,174.670,40.948,157.968
C05281=1052.644,405.951,375.709,174.662,40.941,157.966
C05282=1052.635,405.704,375.754,174.653,40.933,157.963
C05283=1052.626,405.459,375.797,174.646,40.925,157.961
C05284=1052.618,405.212,375.842,174.638,40.918,157.959
C05285=1052.610,404.967,375.886,174.631,40.910,157.956
C05286=1052.600,404.721,375.931,174.623,40.902,157.954
C05287=1052.591,404.475,375.974,174.615,40.895,157.952
C05288=1052.583,404.229,376.019,174.607,40.888,157.949
C05289=1052.574,403.983,376.063,174.599,40.880,157.947
C05290=1052.562,403.621,376.128,174.588,40.868,157.944
C05291=1052.548,403.258,376.193,174.577,40.858,157.940
C05292=1052.535,402.896,376.257,174.566,40.846,157.937
C05293=1052.523,402.534,376.321,174.554,40.836,157.934
C05294=1052.514,402.288,376.365,174.547,40.828,157.931
C05295=1052.506,402.043,376.409,174.539,40.821,157.929
C05296=1052.496,401.796,376.452,174.532,40.813,157.927
C05297=1052.488,401.550,376.497,174.524,40.806,157.925
C05298=1052.480,401.304,376.540,174.517,40.799,157.922
C05299=1052.470,401.058,376.584,174.510,40.791,157.920
C05300=1052.462,400.812,376.627,174.502,40.784,157.918
C05301=1052.453,400.566,376.670,174.495,40.776,157.916
C05302=1052.445,400.321,376.713,174.487,40.769,157.914
C05303=1052.436,400.074,376.757,174.480,40.762,157.911
C05304=1052.428,399.827,376.801,174.472,40.755,157.909
C05305=1052.419,399.582,376.844,174.465,40.748,157.907
C05306=1052.410,399.336,376.887,174.458,40.740,157.905
C05307=1052.402,399.090,376.930,174.450,40.733,157.903
C05308=1052.393,398.844,376.973,174.443,40.726,157.901
C05309=1052.385,398.598,377.016,174.436,40.719,157.898
C05310=1052.376,398.352,377.059,174.428,40.712,157.896
C05311=1052.368,398.106,377.102,174.422,40.705,157.894
C05312=1052.359,397.860,377.146,174.415,40.698,157.892
C05313=1052.351,397.614,377.189,174.407,40.691,157.890
C05314=1052.342,397.368,377.232,174.400,40.683,157.888
C05315=1052.334,397.121,377.275,174.393,40.677,157.886
C05316=1052.325,396.875,377.318,174.385,40.669,157.884
C05317=1052.317,396.629,377.361,174.378,40.663,157.882
C05318=1052.308,396.383,377.404,174.372,40.655,157.879
C05319=1052.300,396.137,377.447,174.365,40.649,157.877
C05320=1052.291,395.891,377.490,174.357,40.641,157.875
C05321=1052.283,395.644,377.532,174.350,40.635,157.873
C05322=1052.275,395.398,377.575,174.343,40.628,157.871
C05323=1052.266,395.152,377.618,174.336,40.621,157.869
C05324=1052.259,394.906,377.660,174.329,40.614,157.867
C05325=1052.249,394.661,377.702,174.322,40.607,157.865
C05326=1052.241,394.415,377.745,174.315,40.601,157.863
C05327=1052.233,394.168,377.788,174.308,40.594,157.861
C05328=1052.224,393.922,377.831,174.302,40.587,157.859
C05329=1052.217,393.676,377.873,174.295,40.580,157.857
C05330=1052.208,393.430,377.916,174.287,40.574,157.855
C05331=1052.200,393.183,377.958,174.280,40.567,157.853
C05332=1052.191,392.937,378.000,174.274,40.560,157.851
C05333=1052.183,392.691,378.042,174.267,40.553,157.849
C05334=1052.175,392.445,378.085,174.260,40.547,157.847
C05335=1052.167,392.198,378.127,174.254,40.540,157.845
C05336=1052.158,391.953,378.169,174.246,40.533,157.843
C05337=1052.150,391.706,378.211,174.239,40.527,157.841
C05338=1052.142,391.460,378.254,174.233,40.520,157.839
C05339=1052.133,391.214,378.295,174.226,40.513,157.837
C05340=1052.125,390.967,378.337,174.219,40.507,157.835
C05341=1052.117,390.722,378.380,174.213,40.500,157.833
C05342=1052.108,390.476,378.422,174.206,40.494,157.831
C05343=1052.100,390.229,378.464,174.200,40.487,157.829
C05344=1052.092,389.983,378.506,174.193,40.481,157.828
C05345=1052.084,389.737,378.548,174.186,40.474,157.826
C05346=1052.072,389.392,378.606,174.177,40.465,157.823
C05347=1052.061,389.049,378.665,174.168,40.456,157.820
C05348=1052.050,388.705,378.723,174.158,40.447,157.818
C05349=1052.038,388.361,378.780,174.149,40.438,157.815
C05350=1052.030,388.114,378.823,174.143,40.432,157.813
C05351=1052.021,387.868,378.864,174.137,40.425,157.811
C05352=1052.013,387.621,378.906,174.130,40.419,157.810
C05353=1052.005,387.375,378.947,174.124,40.413,157.808
C05354=1051.997,387.129,378.989,174.117,40.407,157.806
C05355=1051.989,386.882,379.030,174.111,40.400,157.804
C05356=1051.981,386.637,379.071,174.104,40.394,157.802
C05357=1051.973,386.389,379.113,174.098,40.388,157.800
C05358=1051.964,386.144,379.154,174.091,40.382,157.799
C05359=1051.956,385.897,379.195,174.085,40.375,157.797
C05360=1051.948,385.651,379.237,174.078,40.369,157.795
C05361=1051.940,385.405,379.278,174.072,40.363,157.793
C05362=1051.932,385.158,379.320,174.065,40.356,157.791
C05363=1051.924,384.912,379.361,174.059,40.351,157.790
C05364=1051.916,384.665,379.401,174.052,40.344,157.788
C05365=1051.908,384.419,379.444,174.046,40.338,157.786
C05366=1051.900,384.172,379.484,174.040,40.332,157.784
C05367=1051.892,383.926,379.525,174.034,40.326,157.782
C05368=1051.884,383.680,379.567,174.028,40.320,157.781
C05369=1051.875,383.433,379.608,174.021,40.314,157.779
C05370=1051.867,383.187,379.648,174.015,40.308,157.777
C05371=1051.860,382.940,379.690,174.008,40.301,157.775
C05372=1051.852,382.694,379.730,174.002,40.296,157.774
C05373=1051.844,382.448,379.771,173.997,40.289,157.772
C05374=1051.836,382.202,379.813,173.990,40.284,157.770
C05375=1051.828,381.955,379.854,173.984,40.277,157.768
C05376=1051.820,381.708,379.895,173.978,40.271,157.767
C05377=1051.812,381.462,379.936,173.971,40.266,157.765
C05378=1051.804,381.216,379.976,173.965,40.259,157.763
C05379=1051.796,380.969,380.017,173.960,40.253,157.761
C05380=1051.789,380.723,380.058,173.954,40.247,157.760
C05381=1051.781,380.476,380.098,173.947,40.241,157.758
C05382=1051.773,380.229,380.139,173.941,40.236,157.756
C05383=1051.766,379.983,380.180,173.936,40.230,157.755
C05384=1051.758,379.737,380.221,173.929,40.224,157.753
C05385=1051.750,379.490,380.261,173.923,40.218,157.751
C05386=1051.742,379.243,380.301,173.917,40.212,157.749
C05387=1051.734,378.996,380.342,173.911,40.206,157.748
C05388=1051.726,378.750,380.383,173.905,40.200,157.746
C05389=1051.718,378.503,380.423,173.899,40.194,157.745
C05390=1051.710,378.257,380.463,173.893,40.189,157.743
C05391=1051.702,378.010,380.503,173.888,40.183,157.741
C05392=1051.694,377.764,380.544,173.881,40.178,157.740
C05393=1051.686,377.517,380.584,173.875,40.172,157.738
C05394=1051.678,377.271,380.625,173.869,40.166,157.736
C05395=1051.671,377.024,380.664,173.864,40.160,157.735
C05396=1051.663,376.778,380.705,173.857,40.154,157.733
C05397=1051.656,376.531,380.745,173.851,40.149,157.732
C05398=1051.648,376.285,380.785,173.846,40.143,157.730
C05399=1051.640,376.038,380.825,173.840,40.137,157.728
C05400=1051.632,375.791,380.865,173.834,40.132,157.727
C05401=1051.624,375.545,380.906,173.829,40.126,157.725
C05402=1051.614,375.233,380.956,173.821,40.119,157.723
C05403=1051.604,374.922,381.006,173.814,40.112,157.721
C05404=1051.595,374.610,381.056,173.806,40.105,157.719
C05405=1051.585,374.298,381.108,173.799,40.098,157.717
C05406=1051.577,374.052,381.147,173.794,40.092,157.715
C05407=1051.569,373.805,381.187,173.787,40.087,157.714
C05408=1051.562,373.558,381.226,173.782,40.081,157.712
C05409=1051.554,373.311,381.266,173.776,40.076,157.711
C05410=1051.547,373.065,381.306,173.770,40.070,157.709
C05411=1051.539,372.818,381.346,173.765,40.065,157.708
C05412=1051.531,372.572,381.386,173.759,40.059,157.706
C05413=1051.524,372.325,381.425,173.753,40.054,157.704
C05414=1051.517,372.078,381.465,173.748,40.048,157.703
C05415=1051.509,371.831,381.505,173.742,40.043,157.701
C05416=1051.502,371.585,381.545,173.737,40.037,157.700
C05417=1051.493,371.338,381.584,173.731,40.032,157.698
C05418=1051.486,371.091,381.624,173.726,40.027,157.697
C05419=1051.478,370.845,381.664,173.720,40.021,157.695
C05420=1051.470,370.598,381.702,173.714,40.015,157.694
C05421=1051.463,370.351,381.742,173.709,40.010,157.692
C05422=1051.454,370.105,381.781,173.703,40.005,157.691
C05423=1051.447,369.858,381.820,173.698,40.000,157.689
C05424=1051.440,369.611,381.860,173.692,39.994,157.688
C05425=1051.432,369.365,381.899,173.687,39.989,157.686
C05426=1051.424,369.117,381.938,173.681,39.984,157.685
C05427=1051.417,368.870,381.978,173.676,39.978,157.683
C05428=1051.409,368.624,382.016,173.670,39.974,157.682
C05429=1051.401,368.377,382.056,173.665,39.968,157.680
C05430=1051.394,368.131,382.095,173.659,39.963,157.679
C05431=1051.386,367.884,382.135,173.654,39.958,157.677
C05432=1051.379,367.637,382.173,173.648,39.952,157.676
C05433=1051.371,367.390,382.213,173.643,39.947,157.674
C05434=1051.364,367.143,382.252,173.637,39.942,157.673
C05435=1051.356,366.897,382.291,173.632,39.937,157.672
C05436=1051.349,366.650,382.330,173.626,39.931,157.670
C05437=1051.341,366.403,382.368,173.621,39.926,157.669
C05438=1051.333,366.157,382.408,173.615,39.921,157.667
C05439=1051.325,365.909,382.446,173.610,39.916,157.666
C05440=1051.319,365.663,382.485,173.604,39.911,157.664
C05441=1051.311,365.415,382.525,173.599,39.906,157.663
C05442=1051.303,365.169,382.563,173.594,39.900,157.661
C05443=1051.296,364.922,382.602,173.589,39.895,157.660
C05444=1051.288,364.675,382.641,173.584,39.890,157.659
C05445=1051.281,364.428,382.680,173.578,39.885,157.657
C05446=1051.274,364.182,382.718,173.573,39.880,157.656
C05447=1051.267,363.934,382.757,173.567,39.875,157.654
C05448=1051.259,363.688,382.795,173.562,39.870,157.653
C05449=1051.252,363.441,382.834,173.557,39.865,157.651
C05450=1051.244,363.194,382.873,173.552,39.860,157.650
C05451=1051.237,362.947,382.912,173.547,39.855,157.649
C05452=1051.229,362.700,382.950,173.541,39.850,157.647
C05453=1051.221,362.453,382.989,173.536,39.845,157.646
C05454=1051.215,362.206,383.027,173.530,39.840,157.644
C05455=1051.207,361.960,383.066,173.526,39.835,157.643
C05456=1051.199,361.713,383.104,173.521,39.830,157.642
C05457=1051.192,361.466,383.143,173.515,39.825,157.640
